C09049=1046.535,19.127,-78.806,170.149,34.517,156.500
C09050=1046.529,18.878,-78.790,170.147,34.515,156.499
C09051=1046.523,18.628,-78.775,170.146,34.514,156.499
C09052=1046.516,18.379,-78.759,170.144,34.512,156.499
C09053=1046.510,18.129,-78.743,170.142,34.511,156.499
C09054=1046.504,17.880,-78.728,170.140,34.509,156.498
C09055=1046.497,17.631,-78.712,170.139,34.508,156.498
C09056=1046.491,17.381,-78.696,170.137,34.506,156.498
C09057=1046.485,17.132,-78.681,170.135,34.505,156.498
C09058=1046.479,16.882,-78.665,170.133,34.503,156.497
C09059=1046.473,16.633,-78.650,170.132,34.502,156.497
C09060=1046.466,16.384,-78.634,170.130,34.500,156.497
C09061=1046.460,16.134,-78.618,170.128,34.499,156.497
C09062=1046.454,15.885,-78.603,170.126,34.497,156.497
C09063=1046.448,15.635,-78.587,170.124,34.495,156.496
C09064=1046.441,15.386,-78.572,170.122,34.494,156.496
C09065=1046.435,15.137,-78.556,170.120,34.493,156.496
C09066=1046.429,14.887,-78.540,170.118,34.491,156.496
C09067=1046.422,14.638,-78.525,170.117,34.489,156.495
C09068=1046.417,14.388,-78.509,170.115,34.488,156.495
C09069=1046.410,14.139,-78.493,170.113,34.486,156.495
C09070=1046.404,13.889,-78.479,170.111,34.485,156.495
C09071=1046.397,13.640,-78.463,170.110,34.484,156.494
C09072=1046.390,13.354,-78.446,170.107,34.482,156.494
C09073=1046.382,13.069,-78.428,170.105,34.480,156.494
C09074=1046.375,12.784,-78.411,170.103,34.478,156.494
C09075=1046.368,12.499,-78.393,170.101,34.477,156.493
C09076=1046.362,12.250,-78.377,170.100,34.476,156.493
C09077=1046.355,12.000,-78.362,170.098,34.474,156.493
C09078=1046.349,11.751,-78.347,170.096,34.472,156.493
C09079=1046.342,11.501,-78.331,170.094,34.471,156.492
C09080=1046.336,11.252,-78.316,170.092,34.470,156.492
C09081=1046.329,11.003,-78.301,170.091,34.468,156.492
C09082=1046.323,10.753,-78.286,170.088,34.467,156.492
C09083=1046.317,10.503,-78.270,170.086,34.466,156.492
C09084=1046.310,10.254,-78.255,170.084,34.464,156.491
C09085=1046.304,10.004,-78.240,170.082,34.462,156.491
C09086=1046.298,9.755,-78.225,170.081,34.461,156.491
C09087=1046.291,9.506,-78.209,170.079,34.460,156.491
C09088=1046.285,9.256,-78.194,170.077,34.458,156.490
C09089=1046.278,9.006,-78.179,170.075,34.457,156.490
C09090=1046.272,8.757,-78.163,170.073,34.456,156.490
C09091=1046.266,8.507,-78.148,170.072,34.454,156.490
C09092=1046.259,8.258,-78.133,170.070,34.452,156.490
C09093=1046.253,8.008,-78.118,170.068,34.451,156.489
C09094=1046.246,7.759,-78.102,170.066,34.450,156.489
C09095=1046.241,7.510,-78.088,170.064,34.448,156.489
C09096=1046.234,7.260,-78.073,170.063,34.447,156.489
C09097=1046.228,7.011,-78.058,170.061,34.446,156.488
C09098=1046.221,6.762,-78.042,170.059,34.444,156.488
C09099=1046.216,6.512,-78.027,170.057,34.442,156.488
C09100=1046.209,6.262,-78.012,170.055,34.441,156.488
C09101=1046.203,6.013,-77.997,170.054,34.440,156.488
C09102=1046.196,5.763,-77.981,170.051,34.438,156.487
C09103=1046.190,5.515,-77.967,170.049,34.437,156.487
C09104=1046.184,5.265,-77.952,170.047,34.435,156.487
C09105=1046.177,5.015,-77.937,170.045,34.433,156.487
C09106=1046.171,4.766,-77.922,170.044,34.432,156.486
C09107=1046.165,4.516,-77.907,170.042,34.431,156.486
C09108=1046.158,4.267,-77.891,170.040,34.429,156.486
C09109=1046.152,4.017,-77.876,170.038,34.428,156.486
C09110=1046.147,3.768,-77.861,170.036,34.427,156.486
C09111=1046.140,3.518,-77.846,170.035,34.425,156.485
C09112=1046.134,3.269,-77.831,170.033,34.423,156.485
C09113=1046.127,3.019,-77.816,170.031,34.422,156.485
C09114=1046.121,2.769,-77.801,170.029,34.421,156.485
C09115=1046.115,2.521,-77.786,170.027,34.419,156.484
C09116=1046.109,2.271,-77.771,170.025,34.418,156.484
C09117=1046.102,2.022,-77.756,170.024,34.417,156.484
C09118=1046.096,1.772,-77.741,170.022,34.415,156.484
C09119=1046.089,1.522,-77.726,170.020,34.413,156.484
C09120=1046.084,1.273,-77.712,170.018,34.412,156.483
C09121=1046.077,1.024,-77.697,170.016,34.410,156.483
C09122=1046.071,0.774,-77.682,170.015,34.409,156.483
C09123=1046.065,0.524,-77.666,170.012,34.408,156.483
C09124=1046.059,0.275,-77.652,170.010,34.406,156.482
C09125=1046.053,0.025,-77.637,170.008,34.404,156.482
C09126=1046.047,-0.224,-77.622,170.006,34.403,156.482
C09127=1046.040,-0.474,-77.607,170.004,34.402,156.482
C09128=1046.035,-0.723,-77.592,170.003,34.400,156.482
C09129=1046.028,-0.972,-77.577,170.001,34.399,156.481
C09130=1046.022,-1.222,-77.562,169.999,34.398,156.481
C09131=1046.015,-1.472,-77.547,169.997,34.396,156.481
C09132=1046.010,-1.721,-77.533,169.995,34.394,156.481
C09133=1046.003,-1.970,-77.518,169.993,34.393,156.480
C09134=1045.997,-2.220,-77.503,169.992,34.392,156.480
C09135=1045.991,-2.469,-77.488,169.990,34.390,156.480
C09136=1045.984,-2.752,-77.471,169.988,34.389,156.480
C09137=1045.977,-3.036,-77.454,169.986,34.387,156.479
C09138=1045.970,-3.318,-77.437,169.984,34.386,156.479
C09139=1045.963,-3.602,-77.421,169.981,34.383,156.479
C09140=1045.957,-3.852,-77.406,169.980,34.382,156.479
C09141=1045.949,-4.101,-77.392,169.978,34.381,156.479
C09142=1045.944,-4.350,-77.377,169.976,34.379,156.478
C09143=1045.938,-4.600,-77.363,169.974,34.379,156.478
C09144=1045.931,-4.850,-77.348,169.972,34.377,156.478
C09145=1045.924,-5.099,-77.333,169.969,34.376,156.478
C09146=1045.918,-5.348,-77.319,169.967,34.375,156.478
C09147=1045.912,-5.598,-77.304,169.966,34.373,156.477
C09148=1045.906,-5.848,-77.290,169.964,34.372,156.477
C09149=1045.899,-6.097,-77.276,169.962,34.371,156.477
C09150=1045.893,-6.346,-77.261,169.960,34.369,156.477
C09151=1045.886,-6.596,-77.246,169.958,34.368,156.477
C09152=1045.879,-6.845,-77.232,169.956,34.366,156.476
C09153=1045.874,-7.095,-77.218,169.954,34.365,156.476
C09154=1045.868,-7.345,-77.203,169.952,34.364,156.476
C09155=1045.861,-7.594,-77.188,169.950,34.362,156.476
C09156=1045.855,-7.843,-77.174,169.949,34.361,156.476
C09157=1045.849,-8.093,-77.160,169.947,34.360,156.475
C09158=1045.842,-8.343,-77.145,169.945,34.358,156.475
C09159=1045.836,-8.591,-77.131,169.943,34.357,156.475
C09160=1045.830,-8.842,-77.116,169.941,34.355,156.475
C09161=1045.823,-9.091,-77.101,169.939,34.354,156.475
C09162=1045.817,-9.340,-77.087,169.937,34.353,156.474
C09163=1045.810,-9.590,-77.072,169.935,34.352,156.474
C09164=1045.804,-9.840,-77.058,169.934,34.351,156.474
C09165=1045.798,-10.089,-77.044,169.932,34.349,156.474
C09166=1045.791,-10.338,-77.029,169.930,34.348,156.474
C09167=1045.786,-10.588,-77.015,169.928,34.347,156.474
C09168=1045.779,-10.838,-77.001,169.926,34.345,156.473
C09169=1045.773,-11.087,-76.987,169.924,34.344,156.473
C09170=1045.767,-11.336,-76.972,169.922,34.342,156.473
C09171=1045.760,-11.586,-76.957,169.920,34.341,156.473
C09172=1045.754,-11.835,-76.944,169.917,34.340,156.473
C09173=1045.748,-12.085,-76.929,169.916,34.338,156.472
C09174=1045.741,-12.335,-76.914,169.914,34.337,156.472
C09175=1045.736,-12.584,-76.900,169.912,34.336,156.472
C09176=1045.729,-12.834,-76.886,169.910,34.334,156.472
C09177=1045.723,-13.083,-76.872,169.908,34.333,156.471
C09178=1045.717,-13.333,-76.857,169.906,34.332,156.471
C09179=1045.711,-13.582,-76.844,169.904,34.330,156.471
C09180=1045.704,-13.832,-76.829,169.902,34.329,156.471
C09181=1045.698,-14.082,-76.815,169.900,34.328,156.471
C09182=1045.692,-14.331,-76.801,169.898,34.327,156.471
C09183=1045.685,-14.580,-76.786,169.896,34.325,156.470
C09184=1045.680,-14.830,-76.772,169.895,34.324,156.470
C09185=1045.673,-15.079,-76.758,169.893,34.323,156.470
C09186=1045.667,-15.329,-76.744,169.891,34.321,156.470
C09187=1045.661,-15.579,-76.730,169.889,34.320,156.470
C09188=1045.655,-15.828,-76.716,169.887,34.318,156.469
C09189=1045.648,-16.078,-76.702,169.885,34.318,156.469
C09190=1045.642,-16.327,-76.687,169.883,34.316,156.469
C09191=1045.635,-16.577,-76.674,169.881,34.315,156.469
C09192=1045.628,-16.826,-76.659,169.879,34.314,156.469
C09193=1045.623,-17.076,-76.645,169.877,34.312,156.468
C09194=1045.616,-17.326,-76.632,169.875,34.311,156.468
C09195=1045.610,-17.574,-76.617,169.873,34.310,156.468
C09196=1045.603,-17.824,-76.604,169.871,34.309,156.468
C09197=1045.598,-18.073,-76.589,169.869,34.307,156.468
C09198=1045.591,-18.323,-76.575,169.868,34.307,156.468
C09199=1045.585,-18.573,-76.562,169.866,34.305,156.468
C09200=1045.577,-18.854,-76.546,169.863,34.304,156.467
C09201=1045.570,-19.136,-76.530,169.861,34.302,156.467
C09202=1045.563,-19.417,-76.514,169.858,34.301,156.467
C09203=1045.556,-19.699,-76.499,169.856,34.300,156.467
C09204=1045.550,-19.949,-76.484,169.854,34.298,156.467
C09205=1045.543,-20.198,-76.471,169.852,34.297,156.466
C09206=1045.537,-20.448,-76.457,169.850,34.296,156.466
C09207=1045.531,-20.697,-76.443,169.848,34.295,156.466
C09208=1045.524,-20.947,-76.429,169.846,34.293,156.466
C09209=1045.518,-21.196,-76.415,169.844,34.292,156.466
C09210=1045.512,-21.446,-76.402,169.842,34.291,156.465
C09211=1045.506,-21.695,-76.387,169.840,34.290,156.465
C09212=1045.499,-21.945,-76.373,169.838,34.289,156.465
C09213=1045.493,-22.195,-76.360,169.836,34.287,156.465
C09214=1045.487,-22.444,-76.346,169.834,34.286,156.465
C09215=1045.480,-22.694,-76.332,169.832,34.284,156.465
C09216=1045.475,-22.943,-76.318,169.830,34.284,156.464
C09217=1045.468,-23.193,-76.304,169.828,34.282,156.464
C09218=1045.462,-23.442,-76.291,169.826,34.281,156.464
C09219=1045.455,-23.692,-76.276,169.825,34.280,156.464
C09220=1045.449,-23.941,-76.263,169.823,34.279,156.464
C09221=1045.443,-24.191,-76.250,169.821,34.277,156.464
C09222=1045.437,-24.441,-76.235,169.819,34.276,156.463
C09223=1045.431,-24.690,-76.222,169.817,34.275,156.463
C09224=1045.425,-24.940,-76.208,169.815,34.274,156.463
C09225=1045.418,-25.189,-76.194,169.813,34.273,156.463
C09226=1045.412,-25.438,-76.181,169.811,34.271,156.463
C09227=1045.406,-25.689,-76.166,169.809,34.270,156.462
C09228=1045.400,-25.938,-76.153,169.807,34.269,156.462
C09229=1045.393,-26.187,-76.140,169.805,34.268,156.462
C09230=1045.387,-26.437,-76.126,169.803,34.266,156.462
C09231=1045.381,-26.687,-76.112,169.801,34.265,156.462
C09232=1045.374,-26.935,-76.098,169.799,34.264,156.462
C09233=1045.368,-27.186,-76.084,169.797,34.263,156.462
C09234=1045.362,-27.435,-76.071,169.795,34.261,156.461
C09235=1045.355,-27.685,-76.057,169.793,34.261,156.461
C09236=1045.349,-27.934,-76.044,169.791,34.259,156.461
C09237=1045.343,-28.183,-76.031,169.789,34.259,156.461
C09238=1045.336,-28.433,-76.017,169.786,34.257,156.461
C09239=1045.330,-28.683,-76.004,169.784,34.256,156.461
C09240=1045.324,-28.932,-75.990,169.782,34.255,156.460
C09241=1045.318,-29.182,-75.976,169.780,34.254,156.460
C09242=1045.311,-29.431,-75.963,169.778,34.253,156.460
C09243=1045.305,-29.681,-75.949,169.776,34.251,156.460
C09244=1045.298,-29.931,-75.936,169.774,34.251,156.460
C09245=1045.292,-30.180,-75.923,169.772,34.249,156.460
C09246=1045.285,-30.430,-75.909,169.770,34.248,156.459
C09247=1045.279,-30.679,-75.896,169.768,34.247,156.459
C09248=1045.273,-30.929,-75.883,169.766,34.246,156.459
C09249=1045.268,-31.179,-75.870,169.764,34.245,156.459
C09250=1045.261,-31.428,-75.856,169.762,34.244,156.459
C09251=1045.255,-31.678,-75.843,169.760,34.242,156.459
C09252=1045.249,-31.927,-75.829,169.758,34.242,156.459
C09253=1045.242,-32.177,-75.816,169.756,34.240,156.458
C09254=1045.235,-32.426,-75.802,169.754,34.239,156.458
C09255=1045.229,-32.675,-75.789,169.752,34.238,156.458
C09256=1045.222,-32.925,-75.776,169.750,34.237,156.458
C09257=1045.216,-33.175,-75.762,169.748,34.236,156.458
C09258=1045.210,-33.425,-75.750,169.746,34.235,156.458
C09259=1045.204,-33.674,-75.736,169.744,34.234,156.458
C09260=1045.198,-33.924,-75.722,169.742,34.232,156.457
C09261=1045.192,-34.173,-75.709,169.740,34.232,156.457
C09262=1045.186,-34.423,-75.696,169.738,34.230,156.457
C09263=1045.179,-34.672,-75.682,169.736,34.229,156.457
C09264=1045.172,-34.953,-75.668,169.733,34.228,156.457
C09265=1045.165,-35.233,-75.653,169.731,34.227,156.457
C09266=1045.158,-35.515,-75.638,169.729,34.225,156.456
C09267=1045.151,-35.795,-75.623,169.726,34.224,156.456
C09268=1045.144,-36.045,-75.610,169.724,34.223,156.456
C09269=1045.138,-36.294,-75.596,169.722,34.222,156.456
C09270=1045.132,-36.544,-75.584,169.720,34.221,156.456
C09271=1045.126,-36.794,-75.571,169.718,34.220,156.456
C09272=1045.120,-37.043,-75.557,169.716,34.219,156.456
C09273=1045.113,-37.293,-75.544,169.714,34.217,156.455
C09274=1045.108,-37.543,-75.531,169.712,34.217,156.455
C09275=1045.102,-37.792,-75.517,169.710,34.215,156.455
C09276=1045.096,-38.042,-75.504,169.708,34.214,156.455
C09277=1045.090,-38.291,-75.492,169.706,34.213,156.455
C09278=1045.083,-38.541,-75.478,169.704,34.212,156.455
C09279=1045.077,-38.791,-75.465,169.702,34.211,156.455
C09280=1045.071,-39.041,-75.452,169.700,34.210,156.454
C09281=1045.064,-39.290,-75.439,169.698,34.209,156.454
C09282=1045.057,-39.539,-75.426,169.696,34.208,156.454
C09283=1045.051,-39.789,-75.413,169.694,34.207,156.454
C09284=1045.045,-40.039,-75.400,169.692,34.206,156.454
C09285=1045.039,-40.289,-75.387,169.689,34.205,156.454
C09286=1045.032,-40.537,-75.375,169.687,34.204,156.454
C09287=1045.026,-40.787,-75.361,169.685,34.203,156.454
C09288=1045.020,-41.037,-75.349,169.683,34.202,156.453
C09289=1045.013,-41.287,-75.335,169.681,34.201,156.453
C09290=1045.007,-41.536,-75.323,169.678,34.200,156.453
C09291=1045.001,-41.786,-75.309,169.676,34.199,156.453
C09292=1044.994,-42.035,-75.297,169.674,34.198,156.453
C09293=1044.988,-42.285,-75.284,169.672,34.197,156.453
C09294=1044.982,-42.534,-75.272,169.670,34.196,156.453
C09295=1044.976,-42.784,-75.258,169.668,34.195,156.453
C09296=1044.969,-43.034,-75.245,169.666,34.194,156.452
C09297=1044.962,-43.283,-75.233,169.663,34.193,156.452
C09298=1044.956,-43.533,-75.219,169.661,34.192,156.452
C09299=1044.950,-43.782,-75.207,169.659,34.191,156.452
C09300=1044.944,-44.032,-75.194,169.657,34.191,156.452
C09301=1044.938,-44.282,-75.181,169.655,34.189,156.452
C09302=1044.932,-44.531,-75.169,169.653,34.188,156.452
C09303=1044.925,-44.780,-75.156,169.651,34.188,156.452
C09304=1044.919,-45.030,-75.143,169.649,34.186,156.451
C09305=1044.913,-45.280,-75.130,169.647,34.185,156.451
C09306=1044.907,-45.529,-75.118,169.645,34.185,156.451
C09307=1044.900,-45.779,-75.104,169.643,34.183,156.451
C09308=1044.894,-46.029,-75.092,169.640,34.183,156.451
C09309=1044.888,-46.279,-75.079,169.638,34.182,156.451
C09310=1044.882,-46.528,-75.066,169.636,34.180,156.451
C09311=1044.875,-46.778,-75.054,169.634,34.180,156.451
C09312=1044.869,-47.027,-75.041,169.632,34.179,156.451
C09313=1044.863,-47.277,-75.028,169.630,34.177,156.450
C09314=1044.857,-47.527,-75.016,169.628,34.177,156.450
C09315=1044.850,-47.776,-75.003,169.626,34.176,156.450
C09316=1044.844,-48.026,-74.991,169.624,34.175,156.450
C09317=1044.838,-48.275,-74.978,169.622,34.174,156.450
C09318=1044.832,-48.525,-74.965,169.619,34.173,156.450
C09319=1044.825,-48.774,-74.953,169.617,34.172,156.450
C09320=1044.819,-49.024,-74.940,169.615,34.171,156.450
C09321=1044.813,-49.273,-74.927,169.613,34.170,156.450
C09322=1044.807,-49.523,-74.914,169.611,34.169,156.449
C09323=1044.801,-49.773,-74.902,169.609,34.168,156.449
C09324=1044.794,-50.022,-74.889,169.607,34.167,156.449
C09325=1044.789,-50.272,-74.877,169.605,34.166,156.449
C09326=1044.782,-50.522,-74.865,169.603,34.165,156.449
C09327=1044.776,-50.771,-74.852,169.600,34.164,156.449
C09328=1044.769,-51.053,-74.838,169.598,34.163,156.449
C09329=1044.761,-51.333,-74.824,169.596,34.163,156.449
C09330=1044.754,-51.615,-74.810,169.593,34.162,156.449
C09331=1044.747,-51.896,-74.796,169.591,34.160,156.448
C09332=1044.741,-52.146,-74.784,169.589,34.160,156.448
C09333=1044.735,-52.396,-74.772,169.586,34.159,156.448
C09334=1044.728,-52.645,-74.760,169.584,34.158,156.448
C09335=1044.722,-52.894,-74.747,169.582,34.157,156.448
C09336=1044.715,-53.144,-74.735,169.580,34.157,156.448
C09337=1044.709,-53.393,-74.723,169.578,34.156,156.448
C09338=1044.703,-53.643,-74.710,169.576,34.155,156.448
C09339=1044.696,-53.893,-74.698,169.573,34.154,156.448
C09340=1044.690,-54.143,-74.686,169.571,34.153,156.448
C09341=1044.684,-54.392,-74.674,169.569,34.153,156.448
C09342=1044.677,-54.642,-74.662,169.567,34.152,156.447
C09343=1044.671,-54.892,-74.649,169.565,34.151,156.447
C09344=1044.664,-55.141,-74.637,169.563,34.150,156.447
C09345=1044.657,-55.390,-74.625,169.560,34.150,156.447
C09346=1044.651,-55.640,-74.612,169.558,34.149,156.447
C09347=1044.645,-55.890,-74.600,169.556,34.148,156.447
C09348=1044.639,-56.140,-74.587,169.554,34.147,156.447
C09349=1044.632,-56.389,-74.576,169.552,34.147,156.447
C09350=1044.626,-56.639,-74.564,169.550,34.146,156.447
C09351=1044.620,-56.889,-74.551,169.547,34.145,156.447
C09352=1044.613,-57.138,-74.539,169.545,34.144,156.447
C09353=1044.606,-57.388,-74.527,169.543,34.143,156.447
C09354=1044.601,-57.637,-74.515,169.541,34.143,156.447
C09355=1044.594,-57.887,-74.503,169.539,34.142,156.446
C09356=1044.589,-58.137,-74.490,169.537,34.141,156.446
C09357=1044.582,-58.386,-74.478,169.534,34.140,156.446
C09358=1044.575,-58.636,-74.466,169.532,34.140,156.446
C09359=1044.570,-58.886,-74.455,169.530,34.139,156.446
C09360=1044.563,-59.136,-74.443,169.528,34.138,156.446
C09361=1044.556,-59.385,-74.431,169.526,34.137,156.446
C09362=1044.551,-59.634,-74.419,169.523,34.136,156.446
C09363=1044.544,-59.884,-74.407,169.521,34.136,156.446
C09364=1044.538,-60.134,-74.395,169.519,34.135,156.446
C09365=1044.532,-60.384,-74.382,169.517,34.134,156.446
C09366=1044.525,-60.633,-74.370,169.515,34.133,156.446
C09367=1044.519,-60.883,-74.358,169.512,34.133,156.445
C09368=1044.513,-61.132,-74.346,169.510,34.132,156.445
C09369=1044.507,-61.382,-74.335,169.508,34.131,156.445
C09370=1044.500,-61.632,-74.323,169.506,34.130,156.445
C09371=1044.494,-61.881,-74.310,169.504,34.130,156.445
C09372=1044.488,-62.131,-74.298,169.502,34.129,156.445
C09373=1044.482,-62.380,-74.287,169.499,34.128,156.445
C09374=1044.476,-62.630,-74.274,169.497,34.127,156.445
C09375=1044.469,-62.880,-74.263,169.495,34.126,156.445
C09376=1044.463,-63.130,-74.251,169.493,34.126,156.445
C09377=1044.457,-63.379,-74.238,169.491,34.125,156.445
C09378=1044.451,-63.628,-74.227,169.488,34.124,156.445
C09379=1044.444,-63.878,-74.215,169.486,34.123,156.445
C09380=1044.438,-64.128,-74.204,169.484,34.123,156.444
C09381=1044.432,-64.378,-74.191,169.482,34.122,156.444
C09382=1044.426,-64.627,-74.179,169.480,34.121,156.444
C09383=1044.419,-64.876,-74.167,169.477,34.120,156.444
C09384=1044.414,-65.127,-74.156,169.475,34.120,156.444
C09385=1044.407,-65.377,-74.144,169.473,34.119,156.444
C09386=1044.401,-65.625,-74.132,169.471,34.119,156.444
C09387=1044.395,-65.875,-74.119,169.469,34.118,156.444
C09388=1044.389,-66.125,-74.108,169.466,34.117,156.444
C09389=1044.383,-66.374,-74.097,169.464,34.116,156.444
C09390=1044.376,-66.624,-74.085,169.462,34.115,156.444
C09391=1044.370,-66.874,-74.073,169.460,34.115,156.444
C09392=1044.364,-67.122,-74.062,169.457,34.114,156.444
C09393=1044.358,-67.370,-74.049,169.455,34.113,156.444
C09394=1044.352,-67.618,-74.038,169.453,34.112,156.443
C09395=1044.346,-67.865,-74.026,169.451,34.112,156.443
C09396=1044.339,-68.113,-74.014,169.449,34.111,156.443
C09397=1044.334,-68.362,-74.003,169.447,34.111,156.443
C09398=1044.327,-68.610,-73.991,169.444,34.110,156.443
C09399=1044.321,-68.857,-73.979,169.442,34.109,156.443
C09400=1044.315,-69.108,-73.968,169.440,34.108,156.443
C09401=1044.309,-69.356,-73.956,169.438,34.108,156.443
C09402=1044.303,-69.607,-73.945,169.435,34.107,156.443
C09403=1044.297,-69.855,-73.933,169.433,34.107,156.443
C09404=1044.291,-70.105,-73.921,169.431,34.106,156.443
C09405=1044.285,-70.356,-73.909,169.429,34.105,156.443
C09406=1044.279,-70.604,-73.898,169.427,34.104,156.443
C09407=1044.272,-70.855,-73.887,169.424,34.103,156.443
C09408=1044.267,-71.104,-73.874,169.422,34.103,156.443
C09409=1044.261,-71.354,-73.863,169.420,34.102,156.442
C09410=1044.254,-71.604,-73.851,169.418,34.102,156.442
C09411=1044.248,-71.853,-73.840,169.415,34.101,156.442
C09412=1044.242,-72.103,-73.828,169.413,34.100,156.442
C09413=1044.237,-72.352,-73.817,169.411,34.099,156.442
C09414=1044.230,-72.602,-73.805,169.409,34.099,156.442
C09415=1044.224,-72.852,-73.794,169.407,34.098,156.442
C09416=1044.218,-73.101,-73.782,169.404,34.098,156.442
C09417=1044.212,-73.352,-73.770,169.402,34.097,156.442
C09418=1044.206,-73.600,-73.759,169.400,34.096,156.442
C09419=1044.200,-73.851,-73.747,169.398,34.095,156.442
C09420=1044.194,-74.099,-73.736,169.395,34.095,156.442
C09421=1044.187,-74.350,-73.725,169.393,34.094,156.442
C09422=1044.181,-74.599,-73.714,169.391,34.094,156.442
C09423=1044.175,-74.849,-73.702,169.389,34.093,156.442
C09424=1044.168,-75.135,-73.688,169.386,34.093,156.442
C09425=1044.161,-75.421,-73.676,169.383,34.092,156.442
C09426=1044.153,-75.707,-73.663,169.381,34.091,156.442
C09427=1044.146,-75.993,-73.650,169.378,34.090,156.442
C09428=1044.140,-76.243,-73.639,169.376,34.090,156.442
C09429=1044.134,-76.493,-73.627,169.374,34.089,156.441
C09430=1044.128,-76.742,-73.616,169.371,34.089,156.442
C09431=1044.121,-76.992,-73.605,169.369,34.088,156.441
C09432=1044.116,-77.241,-73.594,169.367,34.088,156.441
C09433=1044.109,-77.491,-73.582,169.365,34.088,156.441
C09434=1044.103,-77.740,-73.571,169.362,34.087,156.441
C09435=1044.097,-77.991,-73.560,169.360,34.086,156.441
C09436=1044.091,-78.240,-73.549,169.358,34.086,156.441
C09437=1044.085,-78.490,-73.537,169.355,34.085,156.441
C09438=1044.079,-78.739,-73.526,169.353,34.085,156.441
C09439=1044.073,-78.989,-73.515,169.351,34.084,156.441
C09440=1044.067,-79.239,-73.504,169.349,34.084,156.441
C09441=1044.060,-79.488,-73.492,169.346,34.083,156.441
C09442=1044.054,-79.738,-73.481,169.344,34.082,156.441
C09443=1044.047,-79.988,-73.470,169.342,34.082,156.441
C09444=1044.042,-80.237,-73.460,169.339,34.081,156.441
C09445=1044.035,-80.488,-73.448,169.337,34.081,156.441
C09446=1044.030,-80.737,-73.437,169.335,34.081,156.441
C09447=1044.022,-80.986,-73.426,169.333,34.080,156.441
C09448=1044.016,-81.236,-73.415,169.330,34.080,156.441
C09449=1044.010,-81.486,-73.404,169.328,34.079,156.441
C09450=1044.004,-81.735,-73.394,169.326,34.079,156.441
C09451=1043.997,-81.985,-73.382,169.324,34.079,156.441
C09452=1043.991,-82.235,-73.371,169.322,34.078,156.441
C09453=1043.984,-82.485,-73.361,169.320,34.078,156.441
C09454=1043.979,-82.734,-73.350,169.317,34.077,156.441
C09455=1043.972,-82.984,-73.339,169.315,34.077,156.441
C09456=1043.965,-83.268,-73.326,169.312,34.076,156.441
C09457=1043.958,-83.554,-73.314,169.310,34.076,156.441
C09458=1043.951,-83.838,-73.301,169.307,34.076,156.441
C09459=1043.944,-84.123,-73.289,169.304,34.075,156.441
C09460=1043.938,-84.373,-73.278,169.302,34.075,156.441
C09461=1043.931,-84.623,-73.267,169.300,34.074,156.441
C09462=1043.925,-84.872,-73.256,169.298,34.074,156.441
C09463=1043.919,-85.122,-73.245,169.295,34.074,156.441
C09464=1043.912,-85.371,-73.235,169.293,34.073,156.441
C09465=1043.907,-85.621,-73.224,169.291,34.073,156.441
C09466=1043.900,-85.871,-73.213,169.288,34.073,156.441
C09467=1043.894,-86.120,-73.202,169.286,34.072,156.441
C09468=1043.887,-86.370,-73.191,169.284,34.072,156.441
C09469=1043.882,-86.620,-73.180,169.281,34.072,156.441
C09470=1043.875,-86.869,-73.170,169.279,34.071,156.441
C09471=1043.869,-87.119,-73.159,169.277,34.071,156.441
C09472=1043.863,-87.369,-73.148,169.274,34.071,156.441
C09473=1043.857,-87.618,-73.138,169.272,34.070,156.441
C09474=1043.850,-87.868,-73.126,169.270,34.070,156.441
C09475=1043.845,-88.118,-73.116,169.267,34.070,156.441
C09476=1043.838,-88.368,-73.106,169.265,34.069,156.441
C09477=1043.832,-88.618,-73.095,169.263,34.069,156.441
C09478=1043.826,-88.867,-73.084,169.260,34.068,156.441
C09479=1043.819,-89.117,-73.073,169.258,34.068,156.441
C09480=1043.813,-89.366,-73.062,169.256,34.068,156.441
C09481=1043.808,-89.616,-73.051,169.253,34.067,156.441
C09482=1043.801,-89.865,-73.041,169.251,34.067,156.441
C09483=1043.795,-90.116,-73.031,169.249,34.066,156.441
C09484=1043.789,-90.365,-73.020,169.246,34.066,156.441
C09485=1043.783,-90.615,-73.010,169.244,34.066,156.441
C09486=1043.777,-90.865,-72.998,169.242,34.065,156.441
C09487=1043.770,-91.114,-72.988,169.239,34.065,156.441
C09488=1043.765,-91.364,-72.978,169.237,34.065,156.441
C09489=1043.758,-91.614,-72.967,169.235,34.065,156.441
C09490=1043.752,-91.863,-72.956,169.232,34.064,156.441
C09491=1043.746,-92.113,-72.945,169.230,34.064,156.441
C09492=1043.740,-92.362,-72.935,169.228,34.064,156.441
C09493=1043.734,-92.613,-72.925,169.225,34.064,156.441
C09494=1043.728,-92.862,-72.914,169.223,34.063,156.441
C09495=1043.721,-93.112,-72.903,169.221,34.063,156.441
C09496=1043.716,-93.361,-72.893,169.218,34.063,156.441
C09497=1043.709,-93.612,-72.883,169.216,34.062,156.441
C09498=1043.703,-93.861,-72.872,169.214,34.062,156.441
C09499=1043.697,-94.111,-72.861,169.211,34.061,156.441
C09500=1043.691,-94.360,-72.851,169.209,34.061,156.441
C09501=1043.686,-94.610,-72.840,169.206,34.061,156.441
C09502=1043.678,-94.860,-72.830,169.204,34.061,156.441
C09503=1043.673,-95.110,-72.820,169.202,34.060,156.441
C09504=1043.667,-95.359,-72.809,169.199,34.060,156.441
C09505=1043.661,-95.609,-72.798,169.197,34.060,156.441
C09506=1043.655,-95.859,-72.788,169.196,34.060,156.441
C09507=1043.648,-96.109,-72.778,169.193,34.060,156.441
C09508=1043.643,-96.358,-72.767,169.191,34.059,156.441
C09509=1043.636,-96.608,-72.757,169.189,34.059,156.441
C09510=1043.631,-96.857,-72.746,169.186,34.058,156.441
C09511=1043.625,-97.107,-72.735,169.184,34.058,156.441
C09512=1043.619,-97.357,-72.726,169.182,34.058,156.441
C09513=1043.612,-97.607,-72.715,169.179,34.058,156.441
C09514=1043.606,-97.857,-72.705,169.177,34.058,156.441
C09515=1043.600,-98.106,-72.695,169.175,34.058,156.441
C09516=1043.594,-98.356,-72.685,169.172,34.058,156.441
C09517=1043.588,-98.605,-72.674,169.170,34.057,156.441
C09518=1043.582,-98.855,-72.665,169.167,34.057,156.441
C09519=1043.575,-99.105,-72.654,169.165,34.057,156.441
C09520=1043.569,-99.392,-72.643,169.162,34.057,156.441
C09521=1043.561,-99.678,-72.631,169.159,34.057,156.441
C09522=1043.554,-99.966,-72.619,169.157,34.057,156.442
C09523=1043.547,-100.253,-72.607,169.154,34.056,156.442
C09524=1043.541,-100.502,-72.597,169.152,34.056,156.442
C09525=1043.535,-100.753,-72.587,169.149,34.056,156.442
C09526=1043.529,-101.002,-72.577,169.147,34.056,156.442
C09527=1043.523,-101.252,-72.567,169.144,34.056,156.442
C09528=1043.516,-101.502,-72.556,169.142,34.056,156.442
C09529=1043.510,-101.752,-72.547,169.140,34.055,156.442
C09530=1043.504,-102.001,-72.536,169.137,34.055,156.442
C09531=1043.498,-102.251,-72.526,169.135,34.055,156.442
C09532=1043.492,-102.501,-72.517,169.133,34.055,156.442
C09533=1043.485,-102.750,-72.506,169.130,34.055,156.442
C09534=1043.479,-103.000,-72.497,169.128,34.055,156.442
C09535=1043.474,-103.249,-72.486,169.125,34.054,156.442
C09536=1043.467,-103.499,-72.476,169.123,34.054,156.442
C09537=1043.461,-103.749,-72.467,169.121,34.054,156.442
C09538=1043.455,-103.998,-72.456,169.118,34.055,156.442
C09539=1043.449,-104.248,-72.446,169.116,34.055,156.442
C09540=1043.443,-104.498,-72.436,169.113,34.054,156.442
C09541=1043.436,-104.748,-72.426,169.111,34.054,156.442
C09542=1043.431,-104.998,-72.416,169.109,34.054,156.442
C09543=1043.424,-105.248,-72.406,169.106,34.054,156.442
C09544=1043.418,-105.497,-72.397,169.104,34.054,156.442
C09545=1043.412,-105.747,-72.386,169.102,34.054,156.442
C09546=1043.406,-105.997,-72.376,169.100,34.054,156.443
C09547=1043.400,-106.246,-72.367,169.098,34.054,156.443
C09548=1043.394,-106.496,-72.356,169.095,34.054,156.443
C09549=1043.388,-106.745,-72.347,169.093,34.054,156.443
C09550=1043.382,-106.996,-72.337,169.090,34.053,156.443
C09551=1043.376,-107.245,-72.327,169.088,34.053,156.443
C09552=1043.370,-107.495,-72.318,169.086,34.054,156.443
C09553=1043.363,-107.744,-72.307,169.083,34.054,156.443
C09554=1043.357,-107.994,-72.298,169.081,34.053,156.443
C09555=1043.351,-108.244,-72.288,169.078,34.053,156.443
C09556=1043.345,-108.494,-72.279,169.076,34.054,156.443
C09557=1043.339,-108.743,-72.269,169.073,34.054,156.443
C09558=1043.333,-108.994,-72.259,169.071,34.053,156.443
C09559=1043.327,-109.243,-72.249,169.069,34.053,156.443
C09560=1043.321,-109.493,-72.239,169.066,34.054,156.443
C09561=1043.314,-109.742,-72.229,169.064,34.054,156.444
C09562=1043.308,-109.992,-72.220,169.061,34.053,156.444
C09563=1043.302,-110.242,-72.210,169.059,34.054,156.444
C09564=1043.296,-110.492,-72.201,169.056,34.054,156.444
C09565=1043.290,-110.742,-72.191,169.054,34.054,156.444
C09566=1043.283,-110.991,-72.182,169.052,34.054,156.444
C09567=1043.277,-111.241,-72.172,169.049,34.054,156.444
C09568=1043.271,-111.490,-72.162,169.047,34.054,156.444
C09569=1043.265,-111.739,-72.153,169.044,34.054,156.444
C09570=1043.260,-111.990,-72.142,169.042,34.054,156.444
C09571=1043.254,-112.239,-72.133,169.039,34.054,156.444
C09572=1043.247,-112.489,-72.123,169.037,34.054,156.444
C09573=1043.241,-112.739,-72.114,169.035,34.054,156.444
C09574=1043.235,-112.989,-72.104,169.032,34.054,156.444
C09575=1043.229,-113.239,-72.095,169.030,34.055,156.445
C09576=1043.223,-113.488,-72.085,169.028,34.054,156.445
C09577=1043.217,-113.738,-72.075,169.026,34.054,156.445
C09578=1043.210,-113.988,-72.066,169.023,34.055,156.445
C09579=1043.204,-114.238,-72.056,169.021,34.055,156.445
C09580=1043.199,-114.487,-72.047,169.019,34.054,156.445
C09581=1043.193,-114.737,-72.038,169.016,34.055,156.445
C09582=1043.186,-114.986,-72.028,169.014,34.055,156.445
C09583=1043.180,-115.236,-72.018,169.011,34.055,156.445
C09584=1043.173,-115.523,-72.008,169.008,34.055,156.445
C09585=1043.166,-115.809,-71.997,169.006,34.056,156.445
C09586=1043.160,-116.094,-71.986,169.003,34.055,156.445
C09587=1043.152,-116.381,-71.976,169.000,34.056,156.446
C09588=1043.146,-116.630,-71.966,168.998,34.056,156.446
C09589=1043.140,-116.880,-71.957,168.995,34.056,156.446
C09590=1043.134,-117.130,-71.947,168.993,34.056,156.446
C09591=1043.128,-117.379,-71.938,168.990,34.056,156.446
C09592=1043.122,-117.630,-71.929,168.988,34.056,156.446
C09593=1043.116,-117.879,-71.919,168.985,34.057,156.446
C09594=1043.110,-118.129,-71.910,168.983,34.057,156.446
C09595=1043.103,-118.379,-71.901,168.980,34.057,156.446
C09596=1043.097,-118.628,-71.891,168.978,34.057,156.446
C09597=1043.091,-118.878,-71.882,168.976,34.057,156.447
C09598=1043.085,-119.128,-71.873,168.973,34.057,156.447
C09599=1043.079,-119.378,-71.864,168.971,34.058,156.447
C09600=1043.073,-119.628,-71.854,168.968,34.058,156.447
C09601=1043.067,-119.877,-71.845,168.966,34.058,156.447
C09602=1043.062,-120.127,-71.836,168.963,34.059,156.447
C09603=1043.055,-120.377,-71.827,168.962,34.058,156.447
C09604=1043.048,-120.626,-71.818,168.959,34.059,156.447
C09605=1043.042,-120.876,-71.808,168.957,34.059,156.447
C09606=1043.037,-121.126,-71.799,168.954,34.059,156.447
C09607=1043.031,-121.376,-71.790,168.952,34.060,156.448
C09608=1043.025,-121.625,-71.780,168.949,34.060,156.448
C09609=1043.018,-121.876,-71.772,168.947,34.060,156.448
C09610=1043.013,-122.125,-71.763,168.945,34.061,156.448
C09611=1043.006,-122.374,-71.753,168.942,34.060,156.448
C09612=1043.000,-122.624,-71.744,168.940,34.061,156.448
C09613=1042.994,-122.875,-71.735,168.937,34.061,156.448
C09614=1042.989,-123.124,-71.726,168.935,34.061,156.448
C09615=1042.982,-123.373,-71.717,168.932,34.062,156.448
C09616=1042.976,-123.624,-71.708,168.930,34.062,156.448
C09617=1042.970,-123.874,-71.698,168.927,34.062,156.449
C09618=1042.965,-124.123,-71.690,168.925,34.062,156.449
C09619=1042.958,-124.373,-71.680,168.922,34.062,156.449
C09620=1042.951,-124.622,-71.671,168.920,34.063,156.449
C09621=1042.946,-124.872,-71.663,168.917,34.063,156.449
C09622=1042.940,-125.122,-71.653,168.915,34.064,156.449
C09623=1042.933,-125.372,-71.645,168.912,34.064,156.449
C09624=1042.927,-125.622,-71.635,168.910,34.064,156.449
C09625=1042.922,-125.872,-71.627,168.907,34.065,156.450
C09626=1042.915,-126.121,-71.618,168.905,34.065,156.450
C09627=1042.909,-126.371,-71.608,168.903,34.065,156.450
C09628=1042.904,-126.621,-71.600,168.901,34.065,156.450
C09629=1042.897,-126.870,-71.591,168.899,34.066,156.450
C09630=1042.891,-127.121,-71.582,168.896,34.066,156.450
C09631=1042.885,-127.370,-71.573,168.894,34.066,156.450
C09632=1042.879,-127.620,-71.565,168.891,34.067,156.450
C09633=1042.873,-127.869,-71.555,168.889,34.067,156.450
C09634=1042.868,-128.119,-71.545,168.886,34.067,156.451
C09635=1042.864,-128.369,-71.536,168.884,34.066,156.450
C09636=1042.860,-128.619,-71.525,168.882,34.065,156.450
C09637=1042.858,-128.869,-71.514,168.880,34.064,156.450
C09638=1042.856,-129.118,-71.501,168.878,34.062,156.450
C09639=1042.856,-129.368,-71.489,168.877,34.059,156.449
C09640=1042.856,-129.619,-71.476,168.875,34.057,156.449
C09641=1042.857,-129.869,-71.462,168.873,34.053,156.449
C09642=1042.858,-130.119,-71.447,168.871,34.049,156.448
C09643=1042.860,-130.369,-71.433,168.870,34.045,156.447
C09644=1042.864,-130.619,-71.417,168.869,34.040,156.446
C09645=1042.869,-130.869,-71.401,168.868,34.036,156.446
C09646=1042.874,-131.120,-71.384,168.867,34.030,156.445
C09647=1042.880,-131.370,-71.367,168.867,34.023,156.444
C09648=1042.529,-131.394,-71.617,168.820,34.211,156.477
C09649=1042.523,-131.144,-71.635,168.821,34.218,156.478
C09650=1042.518,-130.894,-71.651,168.821,34.223,156.479
C09651=1042.512,-130.644,-71.667,168.822,34.228,156.479
C09652=1042.510,-130.392,-71.683,168.823,34.233,156.480
C09653=1042.507,-130.143,-71.697,168.824,34.237,156.481
C09654=1042.505,-129.893,-71.712,168.827,34.241,156.482
C09655=1042.504,-129.643,-71.726,168.828,34.244,156.482
C09656=1042.504,-129.392,-71.739,168.830,34.247,156.483
C09657=1042.505,-129.143,-71.752,168.831,34.250,156.483
C09658=1042.506,-128.893,-71.764,168.833,34.251,156.483
C09659=1042.509,-128.642,-71.776,168.835,34.253,156.483
C09660=1042.512,-128.392,-71.787,168.837,34.254,156.484
C09661=1042.516,-128.143,-71.797,168.840,34.255,156.484
C09662=1042.522,-127.893,-71.806,168.842,34.255,156.484
C09663=1042.527,-127.644,-71.815,168.844,34.254,156.483
C09664=1042.533,-127.394,-71.824,168.847,34.254,156.483
C09665=1042.539,-127.144,-71.833,168.849,34.254,156.483
C09666=1042.546,-126.895,-71.842,168.852,34.254,156.483
C09667=1042.551,-126.644,-71.851,168.854,34.253,156.483
C09668=1042.558,-126.395,-71.860,168.857,34.253,156.483
C09669=1042.564,-126.145,-71.868,168.859,34.252,156.483
C09670=1042.570,-125.895,-71.878,168.861,34.252,156.483
C09671=1042.576,-125.645,-71.887,168.863,34.252,156.482
C09672=1042.582,-125.396,-71.895,168.866,34.251,156.482
C09673=1042.588,-125.146,-71.905,168.868,34.251,156.482
C09674=1042.594,-124.896,-71.914,168.871,34.250,156.482
C09675=1042.600,-124.647,-71.922,168.873,34.250,156.482
C09676=1042.606,-124.397,-71.931,168.876,34.250,156.482
C09677=1042.612,-124.147,-71.941,168.878,34.249,156.482
C09678=1042.618,-123.897,-71.949,168.881,34.249,156.482
C09679=1042.625,-123.648,-71.958,168.883,34.249,156.482
C09680=1042.631,-123.398,-71.968,168.886,34.249,156.481
C09681=1042.637,-123.148,-71.976,168.888,34.248,156.481
C09682=1042.642,-122.899,-71.986,168.891,34.248,156.481
C09683=1042.648,-122.649,-71.995,168.893,34.248,156.481
C09684=1042.655,-122.399,-72.004,168.896,34.247,156.481
C09685=1042.661,-122.149,-72.013,168.898,34.247,156.481
C09686=1042.667,-121.900,-72.022,168.901,34.247,156.481
C09687=1042.673,-121.649,-72.031,168.903,34.246,156.481
C09688=1042.679,-121.400,-72.041,168.906,34.247,156.481
C09689=1042.685,-121.150,-72.050,168.908,34.246,156.480
C09690=1042.691,-120.901,-72.059,168.910,34.245,156.480
C09691=1042.697,-120.651,-72.068,168.913,34.246,156.480
C09692=1042.703,-120.401,-72.077,168.915,34.245,156.480
C09693=1042.709,-120.151,-72.087,168.918,34.245,156.480
C09694=1042.715,-119.901,-72.096,168.920,34.245,156.480
C09695=1042.721,-119.651,-72.105,168.922,34.244,156.480
C09696=1042.727,-119.402,-72.114,168.924,34.244,156.480
C09697=1042.734,-119.152,-72.123,168.927,34.244,156.480
C09698=1042.740,-118.902,-72.133,168.929,34.244,156.480
C09699=1042.746,-118.652,-72.142,168.932,34.244,156.479
C09700=1042.752,-118.403,-72.151,168.934,34.243,156.479
C09701=1042.758,-118.153,-72.161,168.937,34.243,156.479
C09702=1042.764,-117.903,-72.170,168.939,34.243,156.479
C09703=1042.770,-117.653,-72.180,168.942,34.243,156.479
C09704=1042.776,-117.404,-72.189,168.944,34.242,156.479
C09705=1042.781,-117.154,-72.198,168.946,34.243,156.479
C09706=1042.788,-116.904,-72.207,168.949,34.242,156.479
C09707=1042.795,-116.655,-72.216,168.951,34.242,156.479
C09708=1042.801,-116.405,-72.226,168.954,34.242,156.479
C09709=1042.807,-116.118,-72.237,168.957,34.242,156.479
C09710=1042.815,-115.833,-72.247,168.960,34.241,156.478
C09711=1042.821,-115.547,-72.258,168.962,34.241,156.478
C09712=1042.828,-115.260,-72.269,168.965,34.241,156.478
C09713=1042.834,-115.010,-72.279,168.968,34.241,156.478
C09714=1042.840,-114.760,-72.288,168.970,34.241,156.478
C09715=1042.847,-114.511,-72.297,168.973,34.240,156.478
C09716=1042.853,-114.261,-72.307,168.975,34.240,156.478
C09717=1042.859,-114.012,-72.316,168.977,34.241,156.478
C09718=1042.864,-113.762,-72.326,168.980,34.240,156.478
C09719=1042.871,-113.512,-72.336,168.982,34.240,156.478
C09720=1042.877,-113.262,-72.345,168.985,34.240,156.477
C09721=1042.883,-113.013,-72.355,168.987,34.240,156.477
C09722=1042.889,-112.763,-72.364,168.989,34.240,156.477
C09723=1042.895,-112.513,-72.374,168.991,34.240,156.477
C09724=1042.901,-112.263,-72.384,168.994,34.240,156.477
C09725=1042.908,-112.013,-72.393,168.996,34.240,156.477
C09726=1042.914,-111.764,-72.403,168.998,34.239,156.477
C09727=1042.920,-111.514,-72.412,169.001,34.239,156.477
C09728=1042.926,-111.265,-72.422,169.003,34.239,156.477
C09729=1042.932,-111.015,-72.431,169.006,34.239,156.477
C09730=1042.938,-110.765,-72.441,169.008,34.239,156.477
C09731=1042.944,-110.516,-72.451,169.011,34.239,156.477
C09732=1042.951,-110.266,-72.460,169.013,34.239,156.477
C09733=1042.956,-110.016,-72.471,169.015,34.239,156.477
C09734=1042.962,-109.766,-72.480,169.018,34.239,156.476
C09735=1042.968,-109.516,-72.490,169.020,34.239,156.476
C09736=1042.975,-109.267,-72.499,169.023,34.239,156.476
C09737=1042.981,-109.017,-72.509,169.025,34.238,156.476
C09738=1042.987,-108.767,-72.518,169.028,34.239,156.476
C09739=1042.993,-108.518,-72.529,169.030,34.239,156.476
C09740=1042.999,-108.268,-72.538,169.033,34.238,156.476
C09741=1043.006,-108.018,-72.548,169.035,34.238,156.476
C09742=1043.012,-107.768,-72.557,169.037,34.238,156.476
C09743=1043.017,-107.518,-72.568,169.040,34.239,156.476
C09744=1043.023,-107.269,-72.577,169.042,34.238,156.476
C09745=1043.030,-107.019,-72.587,169.045,34.238,156.476
C09746=1043.036,-106.770,-72.597,169.047,34.238,156.476
C09747=1043.042,-106.520,-72.607,169.050,34.239,156.476
C09748=1043.048,-106.270,-72.617,169.052,34.239,156.476
C09749=1043.054,-106.020,-72.627,169.054,34.238,156.475
C09750=1043.060,-105.771,-72.637,169.057,34.238,156.475
C09751=1043.067,-105.521,-72.646,169.059,34.238,156.475
C09752=1043.072,-105.271,-72.656,169.062,34.239,156.475
C09753=1043.078,-105.022,-72.667,169.064,34.239,156.475
C09754=1043.085,-104.772,-72.676,169.066,34.239,156.475
C09755=1043.091,-104.522,-72.686,169.068,34.238,156.475
C09756=1043.097,-104.273,-72.697,169.070,34.239,156.475
C09757=1043.103,-104.022,-72.707,169.073,34.239,156.475
C09758=1043.109,-103.772,-72.716,169.075,34.239,156.475
C09759=1043.116,-103.523,-72.726,169.077,34.239,156.475
C09760=1043.121,-103.273,-72.737,169.080,34.239,156.475
C09761=1043.128,-103.023,-72.746,169.082,34.239,156.475
C09762=1043.134,-102.774,-72.756,169.085,34.239,156.475
C09763=1043.139,-102.524,-72.767,169.087,34.239,156.475
C09764=1043.146,-102.275,-72.777,169.090,34.239,156.475
C09765=1043.152,-102.025,-72.786,169.092,34.239,156.475
C09766=1043.158,-101.775,-72.796,169.094,34.239,156.475
C09767=1043.164,-101.526,-72.807,169.097,34.240,156.475
C09768=1043.170,-101.276,-72.816,169.099,34.240,156.475
C09769=1043.177,-101.026,-72.827,169.102,34.240,156.475
C09770=1043.183,-100.776,-72.837,169.104,34.240,156.475
C09771=1043.189,-100.527,-72.848,169.106,34.240,156.475
C09772=1043.195,-100.277,-72.857,169.109,34.240,156.474
C09773=1043.202,-99.989,-72.869,169.111,34.240,156.474
C09774=1043.210,-99.702,-72.881,169.114,34.240,156.474
C09775=1043.216,-99.416,-72.892,169.117,34.240,156.474
C09776=1043.223,-99.129,-72.904,169.120,34.240,156.474
C09777=1043.229,-98.879,-72.914,169.122,34.240,156.474
C09778=1043.236,-98.629,-72.925,169.125,34.241,156.474
C09779=1043.242,-98.379,-72.935,169.127,34.241,156.474
C09780=1043.248,-98.130,-72.945,169.129,34.241,156.474
C09781=1043.254,-97.880,-72.955,169.132,34.241,156.474
C09782=1043.260,-97.631,-72.965,169.134,34.241,156.474
C09783=1043.267,-97.380,-72.975,169.136,34.241,156.474
C09784=1043.273,-97.131,-72.986,169.139,34.241,156.474
C09785=1043.279,-96.881,-72.997,169.141,34.242,156.474
C09786=1043.285,-96.631,-73.007,169.144,34.242,156.474
C09787=1043.290,-96.382,-73.018,169.146,34.242,156.474
C09788=1043.297,-96.132,-73.027,169.148,34.243,156.474
C09789=1043.303,-95.882,-73.038,169.151,34.243,156.474
C09790=1043.309,-95.633,-73.049,169.153,34.243,156.474
C09791=1043.315,-95.383,-73.059,169.155,34.243,156.474
C09792=1043.321,-95.133,-73.069,169.158,34.244,156.474
C09793=1043.327,-94.884,-73.080,169.160,34.244,156.474
C09794=1043.332,-94.634,-73.090,169.162,34.244,156.474
C09795=1043.340,-94.384,-73.101,169.165,34.244,156.474
C09796=1043.345,-94.134,-73.112,169.166,34.244,156.474
C09797=1043.351,-93.885,-73.121,169.169,34.245,156.474
C09798=1043.357,-93.635,-73.132,169.171,34.245,156.474
C09799=1043.363,-93.385,-73.143,169.173,34.245,156.474
C09800=1043.370,-93.136,-73.154,169.176,34.246,156.474
C09801=1043.375,-92.886,-73.164,169.178,34.246,156.474
C09802=1043.382,-92.636,-73.174,169.180,34.246,156.474
C09803=1043.388,-92.386,-73.185,169.183,34.247,156.474
C09804=1043.394,-92.137,-73.196,169.185,34.247,156.474
C09805=1043.400,-91.887,-73.206,169.187,34.247,156.474
C09806=1043.406,-91.638,-73.217,169.190,34.247,156.474
C09807=1043.413,-91.388,-73.227,169.192,34.248,156.474
C09808=1043.419,-91.138,-73.238,169.194,34.248,156.474
C09809=1043.424,-90.888,-73.248,169.197,34.248,156.474
C09810=1043.431,-90.639,-73.259,169.199,34.248,156.474
C09811=1043.437,-90.389,-73.270,169.201,34.248,156.474
C09812=1043.443,-90.139,-73.281,169.204,34.249,156.474
C09813=1043.449,-89.890,-73.291,169.206,34.249,156.474
C09814=1043.456,-89.640,-73.302,169.209,34.250,156.474
C09815=1043.462,-89.390,-73.312,169.211,34.250,156.474
C09816=1043.467,-89.141,-73.323,169.213,34.250,156.474
C09817=1043.474,-88.890,-73.334,169.216,34.251,156.474
C09818=1043.480,-88.641,-73.344,169.218,34.251,156.474
C09819=1043.486,-88.392,-73.355,169.220,34.251,156.474
C09820=1043.492,-88.141,-73.366,169.223,34.252,156.474
C09821=1043.499,-87.892,-73.377,169.225,34.252,156.474
C09822=1043.505,-87.643,-73.388,169.227,34.252,156.474
C09823=1043.511,-87.393,-73.399,169.230,34.253,156.474
C09824=1043.517,-87.143,-73.409,169.232,34.253,156.474
C09825=1043.523,-86.893,-73.419,169.234,34.253,156.474
C09826=1043.529,-86.643,-73.430,169.237,34.253,156.474
C09827=1043.536,-86.394,-73.441,169.239,34.254,156.474
C09828=1043.542,-86.144,-73.452,169.241,34.254,156.474
C09829=1043.548,-85.894,-73.463,169.244,34.254,156.474
C09830=1043.554,-85.645,-73.473,169.246,34.255,156.474
C09831=1043.560,-85.395,-73.484,169.248,34.255,156.474
C09832=1043.566,-85.145,-73.495,169.251,34.255,156.474
C09833=1043.573,-84.896,-73.506,169.253,34.256,156.474
C09834=1043.579,-84.646,-73.517,169.255,34.256,156.474
C09835=1043.585,-84.397,-73.528,169.258,34.256,156.474
C09836=1043.592,-84.147,-73.538,169.260,34.257,156.474
C09837=1043.599,-83.863,-73.551,169.263,34.257,156.474
C09838=1043.606,-83.577,-73.563,169.265,34.257,156.474
C09839=1043.613,-83.293,-73.575,169.268,34.258,156.474
C09840=1043.621,-83.008,-73.588,169.271,34.258,156.474
C09841=1043.626,-82.758,-73.599,169.273,34.259,156.474
C09842=1043.633,-82.508,-73.610,169.275,34.259,156.474
C09843=1043.638,-82.259,-73.621,169.278,34.259,156.474
C09844=1043.645,-82.009,-73.632,169.280,34.260,156.474
C09845=1043.651,-81.759,-73.643,169.282,34.260,156.474
C09846=1043.658,-81.509,-73.654,169.285,34.261,156.474
C09847=1043.664,-81.260,-73.664,169.287,34.261,156.474
C09848=1043.671,-81.010,-73.676,169.289,34.261,156.474
C09849=1043.676,-80.761,-73.687,169.291,34.262,156.474
C09850=1043.683,-80.511,-73.698,169.294,34.262,156.474
C09851=1043.689,-80.262,-73.709,169.296,34.262,156.474
C09852=1043.696,-80.011,-73.720,169.298,34.263,156.474
C09853=1043.701,-79.762,-73.731,169.301,34.263,156.474
C09854=1043.708,-79.512,-73.743,169.303,34.264,156.474
C09855=1043.714,-79.263,-73.754,169.305,34.264,156.474
C09856=1043.720,-79.013,-73.765,169.308,34.265,156.474
C09857=1043.726,-78.763,-73.776,169.310,34.265,156.474
C09858=1043.733,-78.513,-73.786,169.312,34.266,156.474
C09859=1043.739,-78.264,-73.798,169.314,34.266,156.474
C09860=1043.745,-78.014,-73.809,169.317,34.267,156.474
C09861=1043.751,-77.765,-73.820,169.319,34.267,156.474
C09862=1043.758,-77.515,-73.832,169.321,34.268,156.474
C09863=1043.764,-77.265,-73.843,169.324,34.269,156.474
C09864=1043.770,-77.015,-73.854,169.326,34.269,156.474
C09865=1043.776,-76.765,-73.865,169.328,34.269,156.474
C09866=1043.782,-76.516,-73.877,169.330,34.270,156.474
C09867=1043.788,-76.266,-73.888,169.333,34.270,156.474
C09868=1043.794,-76.017,-73.899,169.334,34.271,156.474
C09869=1043.801,-75.767,-73.911,169.336,34.271,156.474
C09870=1043.807,-75.518,-73.922,169.339,34.272,156.474
C09871=1043.813,-75.267,-73.933,169.341,34.272,156.474
C09872=1043.820,-75.018,-73.945,169.343,34.273,156.474
C09873=1043.825,-74.768,-73.956,169.345,34.273,156.474
C09874=1043.832,-74.519,-73.968,169.348,34.274,156.474
C09875=1043.838,-74.269,-73.979,169.350,34.275,156.475
C09876=1043.844,-74.019,-73.990,169.352,34.275,156.475
C09877=1043.850,-73.770,-74.002,169.354,34.276,156.475
C09878=1043.856,-73.520,-74.013,169.357,34.276,156.475
C09879=1043.863,-73.271,-74.025,169.359,34.277,156.475
C09880=1043.868,-73.021,-74.036,169.361,34.277,156.475
C09881=1043.875,-72.771,-74.048,169.363,34.278,156.475
C09882=1043.880,-72.522,-74.059,169.366,34.279,156.475
C09883=1043.887,-72.272,-74.071,169.368,34.280,156.475
C09884=1043.892,-72.022,-74.083,169.370,34.280,156.475
C09885=1043.899,-71.773,-74.095,169.372,34.280,156.475
C09886=1043.905,-71.523,-74.106,169.375,34.281,156.475
C09887=1043.911,-71.274,-74.117,169.377,34.282,156.475
C09888=1043.917,-71.023,-74.129,169.379,34.283,156.475
C09889=1043.923,-70.774,-74.141,169.381,34.284,156.475
C09890=1043.929,-70.524,-74.152,169.384,34.284,156.475
C09891=1043.936,-70.275,-74.164,169.386,34.285,156.475
C09892=1043.941,-70.025,-74.176,169.388,34.285,156.475
C09893=1043.947,-69.775,-74.187,169.390,34.286,156.476
C09894=1043.953,-69.526,-74.199,169.392,34.287,156.476
C09895=1043.960,-69.276,-74.210,169.395,34.287,156.476
C09896=1043.966,-69.026,-74.223,169.397,34.288,156.476
C09897=1043.971,-68.777,-74.234,169.399,34.288,156.476
C09898=1043.978,-68.527,-74.246,169.401,34.289,156.476
C09899=1043.985,-68.278,-74.258,169.404,34.290,156.476
C09900=1043.990,-68.028,-74.269,169.406,34.291,156.476
C09901=1043.997,-67.745,-74.283,169.408,34.292,156.476
C09902=1044.004,-67.462,-74.296,169.411,34.292,156.476
C09903=1044.011,-67.180,-74.309,169.413,34.293,156.476
C09904=1044.018,-66.898,-74.323,169.416,34.294,156.476
C09905=1044.024,-66.647,-74.334,169.418,34.294,156.476
C09906=1044.030,-66.399,-74.346,169.420,34.295,156.476
C09907=1044.037,-66.149,-74.358,169.423,34.296,156.476
C09908=1044.043,-65.898,-74.370,169.425,34.296,156.477
C09909=1044.049,-65.649,-74.382,169.427,34.297,156.477
C09910=1044.055,-65.400,-74.393,169.429,34.298,156.477
C09911=1044.061,-65.150,-74.406,169.431,34.299,156.477
C09912=1044.067,-64.900,-74.417,169.434,34.299,156.477
C09913=1044.074,-64.651,-74.429,169.436,34.300,156.477
C09914=1044.080,-64.402,-74.440,169.438,34.300,156.477
C09915=1044.086,-64.152,-74.453,169.440,34.301,156.477
C09916=1044.092,-63.901,-74.464,169.442,34.302,156.477
C09917=1044.098,-63.653,-74.476,169.445,34.303,156.477
C09918=1044.104,-63.403,-74.488,169.447,34.303,156.477
C09919=1044.111,-63.153,-74.500,169.449,34.304,156.477
C09920=1044.118,-62.904,-74.512,169.451,34.305,156.477
C09921=1044.123,-62.653,-74.524,169.454,34.306,156.477
C09922=1044.129,-62.404,-74.536,169.456,34.306,156.478
C09923=1044.136,-62.155,-74.548,169.458,34.307,156.478
C09924=1044.142,-61.905,-74.560,169.460,34.307,156.478
C09925=1044.149,-61.655,-74.572,169.462,34.308,156.478
C09926=1044.155,-61.406,-74.584,169.465,34.309,156.478
C09927=1044.160,-61.156,-74.596,169.467,34.310,156.478
C09928=1044.167,-60.906,-74.608,169.469,34.310,156.478
C09929=1044.173,-60.657,-74.620,169.472,34.311,156.478
C09930=1044.179,-60.407,-74.632,169.474,34.312,156.478
C09931=1044.186,-60.157,-74.644,169.477,34.313,156.478
C09932=1044.193,-59.908,-74.656,169.479,34.313,156.478
C09933=1044.198,-59.658,-74.668,169.481,34.314,156.478
C09934=1044.205,-59.409,-74.680,169.483,34.315,156.478
C09935=1044.211,-59.159,-74.692,169.485,34.316,156.479
C09936=1044.217,-58.909,-74.704,169.487,34.317,156.479
C09937=1044.224,-58.659,-74.716,169.490,34.317,156.479
C09938=1044.230,-58.410,-74.728,169.492,34.317,156.479
C09939=1044.236,-58.160,-74.740,169.494,34.318,156.479
C09940=1044.242,-57.911,-74.752,169.496,34.319,156.479
C09941=1044.249,-57.661,-74.764,169.498,34.320,156.479
C09942=1044.255,-57.411,-74.777,169.501,34.321,156.479
C09943=1044.261,-57.162,-74.789,169.503,34.321,156.479
C09944=1044.268,-56.912,-74.801,169.505,34.322,156.479
C09945=1044.278,-56.496,-74.821,169.509,34.324,156.479
C09946=1044.289,-56.080,-74.842,169.512,34.324,156.479
C09947=1044.300,-55.664,-74.861,169.516,34.326,156.480
C09948=1044.310,-55.248,-74.882,169.520,34.327,156.480
C09949=1044.317,-54.998,-74.894,169.522,34.328,156.480
C09950=1044.323,-54.748,-74.907,169.524,34.329,156.480
C09951=1044.329,-54.499,-74.919,169.526,34.330,156.480
C09952=1044.335,-54.249,-74.931,169.528,34.330,156.480
C09953=1044.342,-53.999,-74.943,169.530,34.331,156.480
C09954=1044.349,-53.750,-74.955,169.533,34.332,156.480
C09955=1044.355,-53.500,-74.968,169.535,34.333,156.480
C09956=1044.361,-53.251,-74.980,169.537,34.333,156.480
C09957=1044.367,-53.001,-74.993,169.539,34.334,156.480
C09958=1044.374,-52.751,-75.005,169.541,34.335,156.481
C09959=1044.381,-52.502,-75.017,169.543,34.336,156.481
C09960=1044.387,-52.252,-75.029,169.546,34.336,156.481
C09961=1044.395,-51.888,-75.047,169.549,34.337,156.481
C09962=1044.405,-51.523,-75.065,169.552,34.339,156.481
C09963=1044.414,-51.159,-75.083,169.555,34.340,156.481
C09964=1044.424,-50.795,-75.102,169.558,34.341,156.481
C09965=1044.430,-50.545,-75.114,169.560,34.342,156.481
C09966=1044.437,-50.296,-75.126,169.563,34.343,156.481
C09967=1044.443,-50.046,-75.139,169.565,34.343,156.482
C09968=1044.449,-49.796,-75.152,169.567,34.344,156.482
C09969=1044.455,-49.547,-75.164,169.569,34.345,156.482
C09970=1044.461,-49.297,-75.176,169.571,34.346,156.482
C09971=1044.467,-49.047,-75.189,169.573,34.347,156.482
C09972=1044.474,-48.798,-75.202,169.575,34.348,156.482
C09973=1044.480,-48.548,-75.215,169.577,34.349,156.482
C09974=1044.486,-48.298,-75.227,169.579,34.350,156.482
C09975=1044.492,-48.049,-75.240,169.582,34.351,156.482
C09976=1044.498,-47.799,-75.253,169.584,34.352,156.483
C09977=1044.504,-47.549,-75.265,169.586,34.353,156.483
C09978=1044.511,-47.300,-75.278,169.588,34.354,156.483
C09979=1044.517,-47.050,-75.290,169.590,34.354,156.483
C09980=1044.523,-46.801,-75.304,169.592,34.356,156.483
C09981=1044.529,-46.551,-75.316,169.594,34.356,156.483
C09982=1044.536,-46.302,-75.328,169.596,34.357,156.483
C09983=1044.542,-46.052,-75.341,169.598,34.358,156.483
C09984=1044.548,-45.803,-75.354,169.601,34.359,156.484
C09985=1044.554,-45.553,-75.367,169.603,34.360,156.484
C09986=1044.561,-45.304,-75.379,169.605,34.361,156.484
C09987=1044.568,-45.054,-75.393,169.607,34.362,156.484
C09988=1044.574,-44.804,-75.405,169.609,34.363,156.484
C09989=1044.579,-44.554,-75.418,169.611,34.364,156.484
C09990=1044.586,-44.305,-75.431,169.613,34.364,156.484
C09991=1044.592,-44.055,-75.443,169.615,34.366,156.484
C09992=1044.599,-43.806,-75.456,169.617,34.367,156.484
C09993=1044.604,-43.556,-75.469,169.619,34.367,156.485
C09994=1044.611,-43.307,-75.482,169.622,34.369,156.485
C09995=1044.617,-43.057,-75.495,169.624,34.370,156.485
C09996=1044.624,-42.808,-75.507,169.626,34.370,156.485
//INST
///DATE 2021/06/17 10:56
///ATTR SC,RW,RJ
////FRAME ROBOT
///GROUP1 RB1
NOP
MOVL C00000 V=800.0 PL=0
MOVL C00001 V=800.0 PL=0
MOVL C00002 V=800.0 PL=0
MOVL C00003 V=800.0 PL=0
MOVL C00004 V=800.0 PL=0
MOVL C00005 V=800.0 PL=0
MOVL C00006 V=800.0 PL=0
MOVL C00007 V=800.0 PL=0
MOVL C00008 V=800.0 PL=0
MOVL C00009 V=800.0 PL=0
MOVL C00010 V=800.0 PL=0
MOVL C00011 V=800.0 PL=0
MOVL C00012 V=800.0 PL=0
MOVL C00013 V=800.0 PL=0
MOVL C00014 V=800.0 PL=0
MOVL C00015 V=800.0 PL=0
MOVL C00016 V=800.0 PL=0
MOVL C00017 V=800.0 PL=0
MOVL C00018 V=800.0 PL=0
MOVL C00019 V=800.0 PL=0
MOVL C00020 V=800.0 PL=0
MOVL C00021 V=800.0 PL=0
MOVL C00022 V=800.0 PL=0
MOVL C00023 V=800.0 PL=0
MOVL C00024 V=800.0 PL=0
MOVL C00025 V=800.0 PL=0
MOVL C00026 V=800.0 PL=0
MOVL C00027 V=800.0 PL=0
MOVL C00028 V=800.0 PL=0
MOVL C00029 V=800.0 PL=0
MOVL C00030 V=800.0 PL=0
MOVL C00031 V=800.0 PL=0
MOVL C00032 V=800.0 PL=0
MOVL C00033 V=800.0 PL=0
MOVL C00034 V=800.0 PL=0
MOVL C00035 V=800.0 PL=0
MOVL C00036 V=800.0 PL=0
MOVL C00037 V=800.0 PL=0
MOVL C00038 V=800.0 PL=0
MOVL C00039 V=800.0 PL=0
MOVL C00040 V=800.0 PL=0
MOVL C00041 V=800.0 PL=0
MOVL C00042 V=800.0 PL=0
MOVL C00043 V=800.0 PL=0
MOVL C00044 V=800.0 PL=0
MOVL C00045 V=800.0 PL=0
MOVL C00046 V=800.0 PL=0
MOVL C00047 V=800.0 PL=0
MOVL C00048 V=800.0 PL=0
MOVL C00049 V=800.0 PL=0
MOVL C00050 V=800.0 PL=0
MOVL C00051 V=800.0 PL=0
MOVL C00052 V=800.0 PL=0
MOVL C00053 V=800.0 PL=0
MOVL C00054 V=800.0 PL=0
MOVL C00055 V=800.0 PL=0
MOVL C00056 V=800.0 PL=0
MOVL C00057 V=800.0 PL=0
MOVL C00058 V=800.0 PL=0
MOVL C00059 V=800.0 PL=0
MOVL C00060 V=800.0 PL=0
MOVL C00061 V=800.0 PL=0
MOVL C00062 V=800.0 PL=0
MOVL C00063 V=800.0 PL=0
MOVL C00064 V=800.0 PL=0
MOVL C00065 V=800.0 PL=0
MOVL C00066 V=800.0 PL=0
MOVL C00067 V=800.0 PL=0
MOVL C00068 V=800.0 PL=0
MOVL C00069 V=800.0 PL=0
MOVL C00070 V=800.0 PL=0
MOVL C00071 V=800.0 PL=0
MOVL C00072 V=800.0 PL=0
MOVL C00073 V=800.0 PL=0
MOVL C00074 V=800.0 PL=0
MOVL C00075 V=800.0 PL=0
MOVL C00076 V=800.0 PL=0
MOVL C00077 V=800.0 PL=0
MOVL C00078 V=800.0 PL=0
MOVL C00079 V=800.0 PL=0
MOVL C00080 V=800.0 PL=0
MOVL C00081 V=800.0 PL=0
MOVL C00082 V=800.0 PL=0
MOVL C00083 V=800.0 PL=0
MOVL C00084 V=800.0 PL=0
MOVL C00085 V=800.0 PL=0
MOVL C00086 V=800.0 PL=0
MOVL C00087 V=800.0 PL=0
MOVL C00088 V=800.0 PL=0
MOVL C00089 V=800.0 PL=0
MOVL C00090 V=800.0 PL=0
MOVL C00091 V=800.0 PL=0
MOVL C00092 V=800.0 PL=0
MOVL C00093 V=800.0 PL=0
MOVL C00094 V=800.0 PL=0
MOVL C00095 V=800.0 PL=0
MOVL C00096 V=800.0 PL=0
MOVL C00097 V=800.0 PL=0
MOVL C00098 V=800.0 PL=0
MOVL C00099 V=800.0 PL=0
MOVL C00100 V=800.0 PL=0
MOVL C00101 V=800.0 PL=0
MOVL C00102 V=800.0 PL=0
MOVL C00103 V=800.0 PL=0
MOVL C00104 V=800.0 PL=0
MOVL C00105 V=800.0 PL=0
MOVL C00106 V=800.0 PL=0
MOVL C00107 V=800.0 PL=0
MOVL C00108 V=800.0 PL=0
MOVL C00109 V=800.0 PL=0
MOVL C00110 V=800.0 PL=0
MOVL C00111 V=800.0 PL=0
MOVL C00112 V=800.0 PL=0
MOVL C00113 V=800.0 PL=0
MOVL C00114 V=800.0 PL=0
MOVL C00115 V=800.0 PL=0
MOVL C00116 V=800.0 PL=0
MOVL C00117 V=800.0 PL=0
MOVL C00118 V=800.0 PL=0
MOVL C00119 V=800.0 PL=0
MOVL C00120 V=800.0 PL=0
MOVL C00121 V=800.0 PL=0
MOVL C00122 V=800.0 PL=0
MOVL C00123 V=800.0 PL=0
MOVL C00124 V=800.0 PL=0
MOVL C00125 V=800.0 PL=0
MOVL C00126 V=800.0 PL=0
MOVL C00127 V=800.0 PL=0
MOVL C00128 V=800.0 PL=0
MOVL C00129 V=800.0 PL=0
MOVL C00130 V=800.0 PL=0
MOVL C00131 V=800.0 PL=0
MOVL C00132 V=800.0 PL=0
MOVL C00133 V=800.0 PL=0
MOVL C00134 V=800.0 PL=0
MOVL C00135 V=800.0 PL=0
MOVL C00136 V=800.0 PL=0
MOVL C00137 V=800.0 PL=0
MOVL C00138 V=800.0 PL=0
MOVL C00139 V=800.0 PL=0
MOVL C00140 V=800.0 PL=0
MOVL C00141 V=800.0 PL=0
MOVL C00142 V=800.0 PL=0
MOVL C00143 V=800.0 PL=0
MOVL C00144 V=800.0 PL=0
MOVL C00145 V=800.0 PL=0
MOVL C00146 V=800.0 PL=0
MOVL C00147 V=800.0 PL=0
MOVL C00148 V=800.0 PL=0
MOVL C00149 V=800.0 PL=0
MOVL C00150 V=800.0 PL=0
MOVL C00151 V=800.0 PL=0
MOVL C00152 V=800.0 PL=0
MOVL C00153 V=800.0 PL=0
MOVL C00154 V=800.0 PL=0
MOVL C00155 V=800.0 PL=0
MOVL C00156 V=800.0 PL=0
MOVL C00157 V=800.0 PL=0
MOVL C00158 V=800.0 PL=0
MOVL C00159 V=800.0 PL=0
MOVL C00160 V=800.0 PL=0
MOVL C00161 V=800.0 PL=0
MOVL C00162 V=800.0 PL=0
MOVL C00163 V=800.0 PL=0
MOVL C00164 V=800.0 PL=0
MOVL C00165 V=800.0 PL=0
MOVL C00166 V=800.0 PL=0
MOVL C00167 V=800.0 PL=0
MOVL C00168 V=800.0 PL=0
MOVL C00169 V=800.0 PL=0
MOVL C00170 V=800.0 PL=0
MOVL C00171 V=800.0 PL=0
MOVL C00172 V=800.0 PL=0
MOVL C00173 V=800.0 PL=0
MOVL C00174 V=800.0 PL=0
MOVL C00175 V=800.0 PL=0
MOVL C00176 V=800.0 PL=0
MOVL C00177 V=800.0 PL=0
MOVL C00178 V=800.0 PL=0
MOVL C00179 V=800.0 PL=0
MOVL C00180 V=800.0 PL=0
MOVL C00181 V=800.0 PL=0
MOVL C00182 V=800.0 PL=0
MOVL C00183 V=800.0 PL=0
MOVL C00184 V=800.0 PL=0
MOVL C00185 V=800.0 PL=0
MOVL C00186 V=800.0 PL=0
MOVL C00187 V=800.0 PL=0
MOVL C00188 V=800.0 PL=0
MOVL C00189 V=800.0 PL=0
MOVL C00190 V=800.0 PL=0
MOVL C00191 V=800.0 PL=0
MOVL C00192 V=800.0 PL=0
MOVL C00193 V=800.0 PL=0
MOVL C00194 V=800.0 PL=0
MOVL C00195 V=800.0 PL=0
MOVL C00196 V=800.0 PL=0
MOVL C00197 V=800.0 PL=0
MOVL C00198 V=800.0 PL=0
MOVL C00199 V=800.0 PL=0
MOVL C00200 V=800.0 PL=0
MOVL C00201 V=800.0 PL=0
MOVL C00202 V=800.0 PL=0
MOVL C00203 V=800.0 PL=0
MOVL C00204 V=800.0 PL=0
MOVL C00205 V=800.0 PL=0
MOVL C00206 V=800.0 PL=0
MOVL C00207 V=800.0 PL=0
MOVL C00208 V=800.0 PL=0
MOVL C00209 V=800.0 PL=0
MOVL C00210 V=800.0 PL=0
MOVL C00211 V=800.0 PL=0
MOVL C00212 V=800.0 PL=0
MOVL C00213 V=800.0 PL=0
MOVL C00214 V=800.0 PL=0
MOVL C00215 V=800.0 PL=0
MOVL C00216 V=800.0 PL=0
MOVL C00217 V=800.0 PL=0
MOVL C00218 V=800.0 PL=0
MOVL C00219 V=800.0 PL=0
MOVL C00220 V=800.0 PL=0
MOVL C00221 V=800.0 PL=0
MOVL C00222 V=800.0 PL=0
MOVL C00223 V=800.0 PL=0
MOVL C00224 V=800.0 PL=0
MOVL C00225 V=800.0 PL=0
MOVL C00226 V=800.0 PL=0
MOVL C00227 V=800.0 PL=0
MOVL C00228 V=800.0 PL=0
MOVL C00229 V=800.0 PL=0
MOVL C00230 V=800.0 PL=0
MOVL C00231 V=800.0 PL=0
MOVL C00232 V=800.0 PL=0
MOVL C00233 V=800.0 PL=0
MOVL C00234 V=800.0 PL=0
MOVL C00235 V=800.0 PL=0
MOVL C00236 V=800.0 PL=0
MOVL C00237 V=800.0 PL=0
MOVL C00238 V=800.0 PL=0
MOVL C00239 V=800.0 PL=0
MOVL C00240 V=800.0 PL=0
MOVL C00241 V=800.0 PL=0
MOVL C00242 V=800.0 PL=0
MOVL C00243 V=800.0 PL=0
MOVL C00244 V=800.0 PL=0
MOVL C00245 V=800.0 PL=0
MOVL C00246 V=800.0 PL=0
MOVL C00247 V=800.0 PL=0
MOVL C00248 V=800.0 PL=0
MOVL C00249 V=800.0 PL=0
MOVL C00250 V=800.0 PL=0
MOVL C00251 V=800.0 PL=0
MOVL C00252 V=800.0 PL=0
MOVL C00253 V=800.0 PL=0
MOVL C00254 V=800.0 PL=0
MOVL C00255 V=800.0 PL=0
MOVL C00256 V=800.0 PL=0
MOVL C00257 V=800.0 PL=0
MOVL C00258 V=800.0 PL=0
MOVL C00259 V=800.0 PL=0
MOVL C00260 V=800.0 PL=0
MOVL C00261 V=800.0 PL=0
MOVL C00262 V=800.0 PL=0
MOVL C00263 V=800.0 PL=0
MOVL C00264 V=800.0 PL=0
MOVL C00265 V=800.0 PL=0
MOVL C00266 V=800.0 PL=0
MOVL C00267 V=800.0 PL=0
MOVL C00268 V=800.0 PL=0
MOVL C00269 V=800.0 PL=0
MOVL C00270 V=800.0 PL=0
MOVL C00271 V=800.0 PL=0
MOVL C00272 V=800.0 PL=0
MOVL C00273 V=800.0 PL=0
MOVL C00274 V=800.0 PL=0
MOVL C00275 V=800.0 PL=0
MOVL C00276 V=800.0 PL=0
MOVL C00277 V=800.0 PL=0
MOVL C00278 V=800.0 PL=0
MOVL C00279 V=800.0 PL=0
MOVL C00280 V=800.0 PL=0
MOVL C00281 V=800.0 PL=0
MOVL C00282 V=800.0 PL=0
MOVL C00283 V=800.0 PL=0
MOVL C00284 V=800.0 PL=0
MOVL C00285 V=800.0 PL=0
MOVL C00286 V=800.0 PL=0
MOVL C00287 V=800.0 PL=0
MOVL C00288 V=800.0 PL=0
MOVL C00289 V=800.0 PL=0
MOVL C00290 V=800.0 PL=0
MOVL C00291 V=800.0 PL=0
MOVL C00292 V=800.0 PL=0
MOVL C00293 V=800.0 PL=0
MOVL C00294 V=800.0 PL=0
MOVL C00295 V=800.0 PL=0
MOVL C00296 V=800.0 PL=0
MOVL C00297 V=800.0 PL=0
MOVL C00298 V=800.0 PL=0
MOVL C00299 V=800.0 PL=0
MOVL C00300 V=800.0 PL=0
MOVL C00301 V=800.0 PL=0
MOVL C00302 V=800.0 PL=0
MOVL C00303 V=800.0 PL=0
MOVL C00304 V=800.0 PL=0
MOVL C00305 V=800.0 PL=0
MOVL C00306 V=800.0 PL=0
MOVL C00307 V=800.0 PL=0
MOVL C00308 V=800.0 PL=0
MOVL C00309 V=800.0 PL=0
MOVL C00310 V=800.0 PL=0
MOVL C00311 V=800.0 PL=0
MOVL C00312 V=800.0 PL=0
MOVL C00313 V=800.0 PL=0
MOVL C00314 V=800.0 PL=0
MOVL C00315 V=800.0 PL=0
MOVL C00316 V=800.0 PL=0
MOVL C00317 V=800.0 PL=0
MOVL C00318 V=800.0 PL=0
MOVL C00319 V=800.0 PL=0
MOVL C00320 V=800.0 PL=0
MOVL C00321 V=800.0 PL=0
MOVL C00322 V=800.0 PL=0
MOVL C00323 V=800.0 PL=0
MOVL C00324 V=800.0 PL=0
MOVL C00325 V=800.0 PL=0
MOVL C00326 V=800.0 PL=0
MOVL C00327 V=800.0 PL=0
MOVL C00328 V=800.0 PL=0
MOVL C00329 V=800.0 PL=0
MOVL C00330 V=800.0 PL=0
MOVL C00331 V=800.0 PL=0
MOVL C00332 V=800.0 PL=0
MOVL C00333 V=800.0 PL=0
MOVL C00334 V=800.0 PL=0
MOVL C00335 V=800.0 PL=0
MOVL C00336 V=800.0 PL=0
MOVL C00337 V=800.0 PL=0
MOVL C00338 V=800.0 PL=0
MOVL C00339 V=800.0 PL=0
MOVL C00340 V=800.0 PL=0
MOVL C00341 V=800.0 PL=0
MOVL C00342 V=800.0 PL=0
MOVL C00343 V=800.0 PL=0
MOVL C00344 V=800.0 PL=0
MOVL C00345 V=800.0 PL=0
MOVL C00346 V=800.0 PL=0
MOVL C00347 V=800.0 PL=0
MOVL C00348 V=800.0 PL=0
MOVL C00349 V=800.0 PL=0
MOVL C00350 V=800.0 PL=0
MOVL C00351 V=800.0 PL=0
MOVL C00352 V=800.0 PL=0
MOVL C00353 V=800.0 PL=0
MOVL C00354 V=800.0 PL=0
MOVL C00355 V=800.0 PL=0
MOVL C00356 V=800.0 PL=0
MOVL C00357 V=800.0 PL=0
MOVL C00358 V=800.0 PL=0
MOVL C00359 V=800.0 PL=0
MOVL C00360 V=800.0 PL=0
MOVL C00361 V=800.0 PL=0
MOVL C00362 V=800.0 PL=0
MOVL C00363 V=800.0 PL=0
MOVL C00364 V=800.0 PL=0
MOVL C00365 V=800.0 PL=0
MOVL C00366 V=800.0 PL=0
MOVL C00367 V=800.0 PL=0
MOVL C00368 V=800.0 PL=0
MOVL C00369 V=800.0 PL=0
MOVL C00370 V=800.0 PL=0
MOVL C00371 V=800.0 PL=0
MOVL C00372 V=800.0 PL=0
MOVL C00373 V=800.0 PL=0
MOVL C00374 V=800.0 PL=0
MOVL C00375 V=800.0 PL=0
MOVL C00376 V=800.0 PL=0
MOVL C00377 V=800.0 PL=0
MOVL C00378 V=800.0 PL=0
MOVL C00379 V=800.0 PL=0
MOVL C00380 V=800.0 PL=0
MOVL C00381 V=800.0 PL=0
MOVL C00382 V=800.0 PL=0
MOVL C00383 V=800.0 PL=0
MOVL C00384 V=800.0 PL=0
MOVL C00385 V=800.0 PL=0
MOVL C00386 V=800.0 PL=0
MOVL C00387 V=800.0 PL=0
MOVL C00388 V=800.0 PL=0
MOVL C00389 V=800.0 PL=0
MOVL C00390 V=800.0 PL=0
MOVL C00391 V=800.0 PL=0
MOVL C00392 V=800.0 PL=0
MOVL C00393 V=800.0 PL=0
MOVL C00394 V=800.0 PL=0
MOVL C00395 V=800.0 PL=0
MOVL C00396 V=800.0 PL=0
MOVL C00397 V=800.0 PL=0
MOVL C00398 V=800.0 PL=0
MOVL C00399 V=800.0 PL=0
MOVL C00400 V=800.0 PL=0
MOVL C00401 V=800.0 PL=0
MOVL C00402 V=800.0 PL=0
MOVL C00403 V=800.0 PL=0
MOVL C00404 V=800.0 PL=0
MOVL C00405 V=800.0 PL=0
MOVL C00406 V=800.0 PL=0
MOVL C00407 V=800.0 PL=0
MOVL C00408 V=800.0 PL=0
MOVL C00409 V=800.0 PL=0
MOVL C00410 V=800.0 PL=0
MOVL C00411 V=800.0 PL=0
MOVL C00412 V=800.0 PL=0
MOVL C00413 V=800.0 PL=0
MOVL C00414 V=800.0 PL=0
MOVL C00415 V=800.0 PL=0
MOVL C00416 V=800.0 PL=0
MOVL C00417 V=800.0 PL=0
MOVL C00418 V=800.0 PL=0
MOVL C00419 V=800.0 PL=0
MOVL C00420 V=800.0 PL=0
MOVL C00421 V=800.0 PL=0
MOVL C00422 V=800.0 PL=0
MOVL C00423 V=800.0 PL=0
MOVL C00424 V=800.0 PL=0
MOVL C00425 V=800.0 PL=0
MOVL C00426 V=800.0 PL=0
MOVL C00427 V=800.0 PL=0
MOVL C00428 V=800.0 PL=0
MOVL C00429 V=800.0 PL=0
MOVL C00430 V=800.0 PL=0
MOVL C00431 V=800.0 PL=0
MOVL C00432 V=800.0 PL=0
MOVL C00433 V=800.0 PL=0
MOVL C00434 V=800.0 PL=0
MOVL C00435 V=800.0 PL=0
MOVL C00436 V=800.0 PL=0
MOVL C00437 V=800.0 PL=0
MOVL C00438 V=800.0 PL=0
MOVL C00439 V=800.0 PL=0
MOVL C00440 V=800.0 PL=0
MOVL C00441 V=800.0 PL=0
MOVL C00442 V=800.0 PL=0
MOVL C00443 V=800.0 PL=0
MOVL C00444 V=800.0 PL=0
MOVL C00445 V=800.0 PL=0
MOVL C00446 V=800.0 PL=0
MOVL C00447 V=800.0 PL=0
MOVL C00448 V=800.0 PL=0
MOVL C00449 V=800.0 PL=0
MOVL C00450 V=800.0 PL=0
MOVL C00451 V=800.0 PL=0
MOVL C00452 V=800.0 PL=0
MOVL C00453 V=800.0 PL=0
MOVL C00454 V=800.0 PL=0
MOVL C00455 V=800.0 PL=0
MOVL C00456 V=800.0 PL=0
MOVL C00457 V=800.0 PL=0
MOVL C00458 V=800.0 PL=0
MOVL C00459 V=800.0 PL=0
MOVL C00460 V=800.0 PL=0
MOVL C00461 V=800.0 PL=0
MOVL C00462 V=800.0 PL=0
MOVL C00463 V=800.0 PL=0
MOVL C00464 V=800.0 PL=0
MOVL C00465 V=800.0 PL=0
MOVL C00466 V=800.0 PL=0
MOVL C00467 V=800.0 PL=0
MOVL C00468 V=800.0 PL=0
MOVL C00469 V=800.0 PL=0
MOVL C00470 V=800.0 PL=0
MOVL C00471 V=800.0 PL=0
MOVL C00472 V=800.0 PL=0
MOVL C00473 V=800.0 PL=0
MOVL C00474 V=800.0 PL=0
MOVL C00475 V=800.0 PL=0
MOVL C00476 V=800.0 PL=0
MOVL C00477 V=800.0 PL=0
MOVL C00478 V=800.0 PL=0
MOVL C00479 V=800.0 PL=0
MOVL C00480 V=800.0 PL=0
MOVL C00481 V=800.0 PL=0
MOVL C00482 V=800.0 PL=0
MOVL C00483 V=800.0 PL=0
MOVL C00484 V=800.0 PL=0
MOVL C00485 V=800.0 PL=0
MOVL C00486 V=800.0 PL=0
MOVL C00487 V=800.0 PL=0
MOVL C00488 V=800.0 PL=0
MOVL C00489 V=800.0 PL=0
MOVL C00490 V=800.0 PL=0
MOVL C00491 V=800.0 PL=0
MOVL C00492 V=800.0 PL=0
MOVL C00493 V=800.0 PL=0
MOVL C00494 V=800.0 PL=0
MOVL C00495 V=800.0 PL=0
MOVL C00496 V=800.0 PL=0
MOVL C00497 V=800.0 PL=0
MOVL C00498 V=800.0 PL=0
MOVL C00499 V=800.0 PL=0
MOVL C00500 V=800.0 PL=0
MOVL C00501 V=800.0 PL=0
MOVL C00502 V=800.0 PL=0
MOVL C00503 V=800.0 PL=0
MOVL C00504 V=800.0 PL=0
MOVL C00505 V=800.0 PL=0
MOVL C00506 V=800.0 PL=0
MOVL C00507 V=800.0 PL=0
MOVL C00508 V=800.0 PL=0
MOVL C00509 V=800.0 PL=0
MOVL C00510 V=800.0 PL=0
MOVL C00511 V=800.0 PL=0
MOVL C00512 V=800.0 PL=0
MOVL C00513 V=800.0 PL=0
MOVL C00514 V=800.0 PL=0
MOVL C00515 V=800.0 PL=0
MOVL C00516 V=800.0 PL=0
MOVL C00517 V=800.0 PL=0
MOVL C00518 V=800.0 PL=0
MOVL C00519 V=800.0 PL=0
MOVL C00520 V=800.0 PL=0
MOVL C00521 V=800.0 PL=0
MOVL C00522 V=800.0 PL=0
MOVL C00523 V=800.0 PL=0
MOVL C00524 V=800.0 PL=0
MOVL C00525 V=800.0 PL=0
MOVL C00526 V=800.0 PL=0
MOVL C00527 V=800.0 PL=0
MOVL C00528 V=800.0 PL=0
MOVL C00529 V=800.0 PL=0
MOVL C00530 V=800.0 PL=0
MOVL C00531 V=800.0 PL=0
MOVL C00532 V=800.0 PL=0
MOVL C00533 V=800.0 PL=0
MOVL C00534 V=800.0 PL=0
MOVL C00535 V=800.0 PL=0
MOVL C00536 V=800.0 PL=0
MOVL C00537 V=800.0 PL=0
MOVL C00538 V=800.0 PL=0
MOVL C00539 V=800.0 PL=0
MOVL C00540 V=800.0 PL=0
MOVL C00541 V=800.0 PL=0
MOVL C00542 V=800.0 PL=0
MOVL C00543 V=800.0 PL=0
MOVL C00544 V=800.0 PL=0
MOVL C00545 V=800.0 PL=0
MOVL C00546 V=800.0 PL=0
MOVL C00547 V=800.0 PL=0
MOVL C00548 V=800.0 PL=0
MOVL C00549 V=800.0 PL=0
MOVL C00550 V=800.0 PL=0
MOVL C00551 V=800.0 PL=0
MOVL C00552 V=800.0 PL=0
MOVL C00553 V=800.0 PL=0
MOVL C00554 V=800.0 PL=0
MOVL C00555 V=800.0 PL=0
MOVL C00556 V=800.0 PL=0
MOVL C00557 V=800.0 PL=0
MOVL C00558 V=800.0 PL=0
MOVL C00559 V=800.0 PL=0
MOVL C00560 V=800.0 PL=0
MOVL C00561 V=800.0 PL=0
MOVL C00562 V=800.0 PL=0
MOVL C00563 V=800.0 PL=0
MOVL C00564 V=800.0 PL=0
MOVL C00565 V=800.0 PL=0
MOVL C00566 V=800.0 PL=0
MOVL C00567 V=800.0 PL=0
MOVL C00568 V=800.0 PL=0
MOVL C00569 V=800.0 PL=0
MOVL C00570 V=800.0 PL=0
MOVL C00571 V=800.0 PL=0
MOVL C00572 V=800.0 PL=0
MOVL C00573 V=800.0 PL=0
MOVL C00574 V=800.0 PL=0
MOVL C00575 V=800.0 PL=0
MOVL C00576 V=800.0 PL=0
MOVL C00577 V=800.0 PL=0
MOVL C00578 V=800.0 PL=0
MOVL C00579 V=800.0 PL=0
MOVL C00580 V=800.0 PL=0
MOVL C00581 V=800.0 PL=0
MOVL C00582 V=800.0 PL=0
MOVL C00583 V=800.0 PL=0
MOVL C00584 V=800.0 PL=0
MOVL C00585 V=800.0 PL=0
MOVL C00586 V=800.0 PL=0
MOVL C00587 V=800.0 PL=0
MOVL C00588 V=800.0 PL=0
MOVL C00589 V=800.0 PL=0
MOVL C00590 V=800.0 PL=0
MOVL C00591 V=800.0 PL=0
MOVL C00592 V=800.0 PL=0
MOVL C00593 V=800.0 PL=0
MOVL C00594 V=800.0 PL=0
MOVL C00595 V=800.0 PL=0
MOVL C00596 V=800.0 PL=0
MOVL C00597 V=800.0 PL=0
MOVL C00598 V=800.0 PL=0
MOVL C00599 V=800.0 PL=0
MOVL C00600 V=800.0 PL=0
MOVL C00601 V=800.0 PL=0
MOVL C00602 V=800.0 PL=0
MOVL C00603 V=800.0 PL=0
MOVL C00604 V=800.0 PL=0
MOVL C00605 V=800.0 PL=0
MOVL C00606 V=800.0 PL=0
MOVL C00607 V=800.0 PL=0
MOVL C00608 V=800.0 PL=0
MOVL C00609 V=800.0 PL=0
MOVL C00610 V=800.0 PL=0
MOVL C00611 V=800.0 PL=0
MOVL C00612 V=800.0 PL=0
MOVL C00613 V=800.0 PL=0
MOVL C00614 V=800.0 PL=0
MOVL C00615 V=800.0 PL=0
MOVL C00616 V=800.0 PL=0
MOVL C00617 V=800.0 PL=0
MOVL C00618 V=800.0 PL=0
MOVL C00619 V=800.0 PL=0
MOVL C00620 V=800.0 PL=0
MOVL C00621 V=800.0 PL=0
MOVL C00622 V=800.0 PL=0
MOVL C00623 V=800.0 PL=0
MOVL C00624 V=800.0 PL=0
MOVL C00625 V=800.0 PL=0
MOVL C00626 V=800.0 PL=0
MOVL C00627 V=800.0 PL=0
MOVL C00628 V=800.0 PL=0
MOVL C00629 V=800.0 PL=0
MOVL C00630 V=800.0 PL=0
MOVL C00631 V=800.0 PL=0
MOVL C00632 V=800.0 PL=0
MOVL C00633 V=800.0 PL=0
MOVL C00634 V=800.0 PL=0
MOVL C00635 V=800.0 PL=0
MOVL C00636 V=800.0 PL=0
MOVL C00637 V=800.0 PL=0
MOVL C00638 V=800.0 PL=0
MOVL C00639 V=800.0 PL=0
MOVL C00640 V=800.0 PL=0
MOVL C00641 V=800.0 PL=0
MOVL C00642 V=800.0 PL=0
MOVL C00643 V=800.0 PL=0
MOVL C00644 V=800.0 PL=0
MOVL C00645 V=800.0 PL=0
MOVL C00646 V=800.0 PL=0
MOVL C00647 V=800.0 PL=0
MOVL C00648 V=800.0 PL=0
MOVL C00649 V=800.0 PL=0
MOVL C00650 V=800.0 PL=0
MOVL C00651 V=800.0 PL=0
MOVL C00652 V=800.0 PL=0
MOVL C00653 V=800.0 PL=0
MOVL C00654 V=800.0 PL=0
MOVL C00655 V=800.0 PL=0
MOVL C00656 V=800.0 PL=0
MOVL C00657 V=800.0 PL=0
MOVL C00658 V=800.0 PL=0
MOVL C00659 V=800.0 PL=0
MOVL C00660 V=800.0 PL=0
MOVL C00661 V=800.0 PL=0
MOVL C00662 V=800.0 PL=0
MOVL C00663 V=800.0 PL=0
MOVL C00664 V=800.0 PL=0
MOVL C00665 V=800.0 PL=0
MOVL C00666 V=800.0 PL=0
MOVL C00667 V=800.0 PL=0
MOVL C00668 V=800.0 PL=0
MOVL C00669 V=800.0 PL=0
MOVL C00670 V=800.0 PL=0
MOVL C00671 V=800.0 PL=0
MOVL C00672 V=800.0 PL=0
MOVL C00673 V=800.0 PL=0
MOVL C00674 V=800.0 PL=0
MOVL C00675 V=800.0 PL=0
MOVL C00676 V=800.0 PL=0
MOVL C00677 V=800.0 PL=0
MOVL C00678 V=800.0 PL=0
MOVL C00679 V=800.0 PL=0
MOVL C00680 V=800.0 PL=0
MOVL C00681 V=800.0 PL=0
MOVL C00682 V=800.0 PL=0
MOVL C00683 V=800.0 PL=0
MOVL C00684 V=800.0 PL=0
MOVL C00685 V=800.0 PL=0
MOVL C00686 V=800.0 PL=0
MOVL C00687 V=800.0 PL=0
MOVL C00688 V=800.0 PL=0
MOVL C00689 V=800.0 PL=0
MOVL C00690 V=800.0 PL=0
MOVL C00691 V=800.0 PL=0
MOVL C00692 V=800.0 PL=0
MOVL C00693 V=800.0 PL=0
MOVL C00694 V=800.0 PL=0
MOVL C00695 V=800.0 PL=0
MOVL C00696 V=800.0 PL=0
MOVL C00697 V=800.0 PL=0
MOVL C00698 V=800.0 PL=0
MOVL C00699 V=800.0 PL=0
MOVL C00700 V=800.0 PL=0
MOVL C00701 V=800.0 PL=0
MOVL C00702 V=800.0 PL=0
MOVL C00703 V=800.0 PL=0
MOVL C00704 V=800.0 PL=0
MOVL C00705 V=800.0 PL=0
MOVL C00706 V=800.0 PL=0
MOVL C00707 V=800.0 PL=0
MOVL C00708 V=800.0 PL=0
MOVL C00709 V=800.0 PL=0
MOVL C00710 V=800.0 PL=0
MOVL C00711 V=800.0 PL=0
MOVL C00712 V=800.0 PL=0
MOVL C00713 V=800.0 PL=0
MOVL C00714 V=800.0 PL=0
MOVL C00715 V=800.0 PL=0
MOVL C00716 V=800.0 PL=0
MOVL C00717 V=800.0 PL=0
MOVL C00718 V=800.0 PL=0
MOVL C00719 V=800.0 PL=0
MOVL C00720 V=800.0 PL=0
MOVL C00721 V=800.0 PL=0
MOVL C00722 V=800.0 PL=0
MOVL C00723 V=800.0 PL=0
MOVL C00724 V=800.0 PL=0
MOVL C00725 V=800.0 PL=0
MOVL C00726 V=800.0 PL=0
MOVL C00727 V=800.0 PL=0
MOVL C00728 V=800.0 PL=0
MOVL C00729 V=800.0 PL=0
MOVL C00730 V=800.0 PL=0
MOVL C00731 V=800.0 PL=0
MOVL C00732 V=800.0 PL=0
MOVL C00733 V=800.0 PL=0
MOVL C00734 V=800.0 PL=0
MOVL C00735 V=800.0 PL=0
MOVL C00736 V=800.0 PL=0
MOVL C00737 V=800.0 PL=0
MOVL C00738 V=800.0 PL=0
MOVL C00739 V=800.0 PL=0
MOVL C00740 V=800.0 PL=0
MOVL C00741 V=800.0 PL=0
MOVL C00742 V=800.0 PL=0
MOVL C00743 V=800.0 PL=0
MOVL C00744 V=800.0 PL=0
MOVL C00745 V=800.0 PL=0
MOVL C00746 V=800.0 PL=0
MOVL C00747 V=800.0 PL=0
MOVL C00748 V=800.0 PL=0
MOVL C00749 V=800.0 PL=0
MOVL C00750 V=800.0 PL=0
MOVL C00751 V=800.0 PL=0
MOVL C00752 V=800.0 PL=0
MOVL C00753 V=800.0 PL=0
MOVL C00754 V=800.0 PL=0
MOVL C00755 V=800.0 PL=0
MOVL C00756 V=800.0 PL=0
MOVL C00757 V=800.0 PL=0
MOVL C00758 V=800.0 PL=0
MOVL C00759 V=800.0 PL=0
MOVL C00760 V=800.0 PL=0
MOVL C00761 V=800.0 PL=0
MOVL C00762 V=800.0 PL=0
MOVL C00763 V=800.0 PL=0
MOVL C00764 V=800.0 PL=0
MOVL C00765 V=800.0 PL=0
MOVL C00766 V=800.0 PL=0
MOVL C00767 V=800.0 PL=0
MOVL C00768 V=800.0 PL=0
MOVL C00769 V=800.0 PL=0
MOVL C00770 V=800.0 PL=0
MOVL C00771 V=800.0 PL=0
MOVL C00772 V=800.0 PL=0
MOVL C00773 V=800.0 PL=0
MOVL C00774 V=800.0 PL=0
MOVL C00775 V=800.0 PL=0
MOVL C00776 V=800.0 PL=0
MOVL C00777 V=800.0 PL=0
MOVL C00778 V=800.0 PL=0
MOVL C00779 V=800.0 PL=0
MOVL C00780 V=800.0 PL=0
MOVL C00781 V=800.0 PL=0
MOVL C00782 V=800.0 PL=0
MOVL C00783 V=800.0 PL=0
MOVL C00784 V=800.0 PL=0
MOVL C00785 V=800.0 PL=0
MOVL C00786 V=800.0 PL=0
MOVL C00787 V=800.0 PL=0
MOVL C00788 V=800.0 PL=0
MOVL C00789 V=800.0 PL=0
MOVL C00790 V=800.0 PL=0
MOVL C00791 V=800.0 PL=0
MOVL C00792 V=800.0 PL=0
MOVL C00793 V=800.0 PL=0
MOVL C00794 V=800.0 PL=0
MOVL C00795 V=800.0 PL=0
MOVL C00796 V=800.0 PL=0
MOVL C00797 V=800.0 PL=0
MOVL C00798 V=800.0 PL=0
MOVL C00799 V=800.0 PL=0
MOVL C00800 V=800.0 PL=0
MOVL C00801 V=800.0 PL=0
MOVL C00802 V=800.0 PL=0
MOVL C00803 V=800.0 PL=0
MOVL C00804 V=800.0 PL=0
MOVL C00805 V=800.0 PL=0
MOVL C00806 V=800.0 PL=0
MOVL C00807 V=800.0 PL=0
MOVL C00808 V=800.0 PL=0
MOVL C00809 V=800.0 PL=0
MOVL C00810 V=800.0 PL=0
MOVL C00811 V=800.0 PL=0
MOVL C00812 V=800.0 PL=0
MOVL C00813 V=800.0 PL=0
MOVL C00814 V=800.0 PL=0
MOVL C00815 V=800.0 PL=0
MOVL C00816 V=800.0 PL=0
MOVL C00817 V=800.0 PL=0
MOVL C00818 V=800.0 PL=0
MOVL C00819 V=800.0 PL=0
MOVL C00820 V=800.0 PL=0
MOVL C00821 V=800.0 PL=0
MOVL C00822 V=800.0 PL=0
MOVL C00823 V=800.0 PL=0
MOVL C00824 V=800.0 PL=0
MOVL C00825 V=800.0 PL=0
MOVL C00826 V=800.0 PL=0
MOVL C00827 V=800.0 PL=0
MOVL C00828 V=800.0 PL=0
MOVL C00829 V=800.0 PL=0
MOVL C00830 V=800.0 PL=0
MOVL C00831 V=800.0 PL=0
MOVL C00832 V=800.0 PL=0
MOVL C00833 V=800.0 PL=0
MOVL C00834 V=800.0 PL=0
MOVL C00835 V=800.0 PL=0
MOVL C00836 V=800.0 PL=0
MOVL C00837 V=800.0 PL=0
MOVL C00838 V=800.0 PL=0
MOVL C00839 V=800.0 PL=0
MOVL C00840 V=800.0 PL=0
MOVL C00841 V=800.0 PL=0
MOVL C00842 V=800.0 PL=0
MOVL C00843 V=800.0 PL=0
MOVL C00844 V=800.0 PL=0
MOVL C00845 V=800.0 PL=0
MOVL C00846 V=800.0 PL=0
MOVL C00847 V=800.0 PL=0
MOVL C00848 V=800.0 PL=0
MOVL C00849 V=800.0 PL=0
MOVL C00850 V=800.0 PL=0
MOVL C00851 V=800.0 PL=0
MOVL C00852 V=800.0 PL=0
MOVL C00853 V=800.0 PL=0
MOVL C00854 V=800.0 PL=0
MOVL C00855 V=800.0 PL=0
MOVL C00856 V=800.0 PL=0
MOVL C00857 V=800.0 PL=0
MOVL C00858 V=800.0 PL=0
MOVL C00859 V=800.0 PL=0
MOVL C00860 V=800.0 PL=0
MOVL C00861 V=800.0 PL=0
MOVL C00862 V=800.0 PL=0
MOVL C00863 V=800.0 PL=0
MOVL C00864 V=800.0 PL=0
MOVL C00865 V=800.0 PL=0
MOVL C00866 V=800.0 PL=0
MOVL C00867 V=800.0 PL=0
MOVL C00868 V=800.0 PL=0
MOVL C00869 V=800.0 PL=0
MOVL C00870 V=800.0 PL=0
MOVL C00871 V=800.0 PL=0
MOVL C00872 V=800.0 PL=0
MOVL C00873 V=800.0 PL=0
MOVL C00874 V=800.0 PL=0
MOVL C00875 V=800.0 PL=0
MOVL C00876 V=800.0 PL=0
MOVL C00877 V=800.0 PL=0
MOVL C00878 V=800.0 PL=0
MOVL C00879 V=800.0 PL=0
MOVL C00880 V=800.0 PL=0
MOVL C00881 V=800.0 PL=0
MOVL C00882 V=800.0 PL=0
MOVL C00883 V=800.0 PL=0
MOVL C00884 V=800.0 PL=0
MOVL C00885 V=800.0 PL=0
MOVL C00886 V=800.0 PL=0
MOVL C00887 V=800.0 PL=0
MOVL C00888 V=800.0 PL=0
MOVL C00889 V=800.0 PL=0
MOVL C00890 V=800.0 PL=0
MOVL C00891 V=800.0 PL=0
MOVL C00892 V=800.0 PL=0
MOVL C00893 V=800.0 PL=0
MOVL C00894 V=800.0 PL=0
MOVL C00895 V=800.0 PL=0
MOVL C00896 V=800.0 PL=0
MOVL C00897 V=800.0 PL=0
MOVL C00898 V=800.0 PL=0
MOVL C00899 V=800.0 PL=0
MOVL C00900 V=800.0 PL=0
MOVL C00901 V=800.0 PL=0
MOVL C00902 V=800.0 PL=0
MOVL C00903 V=800.0 PL=0
MOVL C00904 V=800.0 PL=0
MOVL C00905 V=800.0 PL=0
MOVL C00906 V=800.0 PL=0
MOVL C00907 V=800.0 PL=0
MOVL C00908 V=800.0 PL=0
MOVL C00909 V=800.0 PL=0
MOVL C00910 V=800.0 PL=0
MOVL C00911 V=800.0 PL=0
MOVL C00912 V=800.0 PL=0
MOVL C00913 V=800.0 PL=0
MOVL C00914 V=800.0 PL=0
MOVL C00915 V=800.0 PL=0
MOVL C00916 V=800.0 PL=0
MOVL C00917 V=800.0 PL=0
MOVL C00918 V=800.0 PL=0
MOVL C00919 V=800.0 PL=0
MOVL C00920 V=800.0 PL=0
MOVL C00921 V=800.0 PL=0
MOVL C00922 V=800.0 PL=0
MOVL C00923 V=800.0 PL=0
MOVL C00924 V=800.0 PL=0
MOVL C00925 V=800.0 PL=0
MOVL C00926 V=800.0 PL=0
MOVL C00927 V=800.0 PL=0
MOVL C00928 V=800.0 PL=0
MOVL C00929 V=800.0 PL=0
MOVL C00930 V=800.0 PL=0
MOVL C00931 V=800.0 PL=0
MOVL C00932 V=800.0 PL=0
MOVL C00933 V=800.0 PL=0
MOVL C00934 V=800.0 PL=0
MOVL C00935 V=800.0 PL=0
MOVL C00936 V=800.0 PL=0
MOVL C00937 V=800.0 PL=0
MOVL C00938 V=800.0 PL=0
MOVL C00939 V=800.0 PL=0
MOVL C00940 V=800.0 PL=0
MOVL C00941 V=800.0 PL=0
MOVL C00942 V=800.0 PL=0
MOVL C00943 V=800.0 PL=0
MOVL C00944 V=800.0 PL=0
MOVL C00945 V=800.0 PL=0
MOVL C00946 V=800.0 PL=0
MOVL C00947 V=800.0 PL=0
MOVL C00948 V=800.0 PL=0
MOVL C00949 V=800.0 PL=0
MOVL C00950 V=800.0 PL=0
MOVL C00951 V=800.0 PL=0
MOVL C00952 V=800.0 PL=0
MOVL C00953 V=800.0 PL=0
MOVL C00954 V=800.0 PL=0
MOVL C00955 V=800.0 PL=0
MOVL C00956 V=800.0 PL=0
MOVL C00957 V=800.0 PL=0
MOVL C00958 V=800.0 PL=0
MOVL C00959 V=800.0 PL=0
MOVL C00960 V=800.0 PL=0
MOVL C00961 V=800.0 PL=0
MOVL C00962 V=800.0 PL=0
MOVL C00963 V=800.0 PL=0
MOVL C00964 V=800.0 PL=0
MOVL C00965 V=800.0 PL=0
MOVL C00966 V=800.0 PL=0
MOVL C00967 V=800.0 PL=0
MOVL C00968 V=800.0 PL=0
MOVL C00969 V=800.0 PL=0
MOVL C00970 V=800.0 PL=0
MOVL C00971 V=800.0 PL=0
MOVL C00972 V=800.0 PL=0
MOVL C00973 V=800.0 PL=0
MOVL C00974 V=800.0 PL=0
MOVL C00975 V=800.0 PL=0
MOVL C00976 V=800.0 PL=0
MOVL C00977 V=800.0 PL=0
MOVL C00978 V=800.0 PL=0
MOVL C00979 V=800.0 PL=0
MOVL C00980 V=800.0 PL=0
MOVL C00981 V=800.0 PL=0
MOVL C00982 V=800.0 PL=0
MOVL C00983 V=800.0 PL=0
MOVL C00984 V=800.0 PL=0
MOVL C00985 V=800.0 PL=0
MOVL C00986 V=800.0 PL=0
MOVL C00987 V=800.0 PL=0
MOVL C00988 V=800.0 PL=0
MOVL C00989 V=800.0 PL=0
MOVL C00990 V=800.0 PL=0
MOVL C00991 V=800.0 PL=0
MOVL C00992 V=800.0 PL=0
MOVL C00993 V=800.0 PL=0
MOVL C00994 V=800.0 PL=0
MOVL C00995 V=800.0 PL=0
MOVL C00996 V=800.0 PL=0
MOVL C00997 V=800.0 PL=0
MOVL C00998 V=800.0 PL=0
MOVL C00999 V=800.0 PL=0
MOVL C01000 V=800.0 PL=0
MOVL C01001 V=800.0 PL=0
MOVL C01002 V=800.0 PL=0
MOVL C01003 V=800.0 PL=0
MOVL C01004 V=800.0 PL=0
MOVL C01005 V=800.0 PL=0
MOVL C01006 V=800.0 PL=0
MOVL C01007 V=800.0 PL=0
MOVL C01008 V=800.0 PL=0
MOVL C01009 V=800.0 PL=0
MOVL C01010 V=800.0 PL=0
MOVL C01011 V=800.0 PL=0
MOVL C01012 V=800.0 PL=0
MOVL C01013 V=800.0 PL=0
MOVL C01014 V=800.0 PL=0
MOVL C01015 V=800.0 PL=0
MOVL C01016 V=800.0 PL=0
MOVL C01017 V=800.0 PL=0
MOVL C01018 V=800.0 PL=0
MOVL C01019 V=800.0 PL=0
MOVL C01020 V=800.0 PL=0
MOVL C01021 V=800.0 PL=0
MOVL C01022 V=800.0 PL=0
MOVL C01023 V=800.0 PL=0
MOVL C01024 V=800.0 PL=0
MOVL C01025 V=800.0 PL=0
MOVL C01026 V=800.0 PL=0
MOVL C01027 V=800.0 PL=0
MOVL C01028 V=800.0 PL=0
MOVL C01029 V=800.0 PL=0
MOVL C01030 V=800.0 PL=0
MOVL C01031 V=800.0 PL=0
MOVL C01032 V=800.0 PL=0
MOVL C01033 V=800.0 PL=0
MOVL C01034 V=800.0 PL=0
MOVL C01035 V=800.0 PL=0
MOVL C01036 V=800.0 PL=0
MOVL C01037 V=800.0 PL=0
MOVL C01038 V=800.0 PL=0
MOVL C01039 V=800.0 PL=0
MOVL C01040 V=800.0 PL=0
MOVL C01041 V=800.0 PL=0
MOVL C01042 V=800.0 PL=0
MOVL C01043 V=800.0 PL=0
MOVL C01044 V=800.0 PL=0
MOVL C01045 V=800.0 PL=0
MOVL C01046 V=800.0 PL=0
MOVL C01047 V=800.0 PL=0
MOVL C01048 V=800.0 PL=0
MOVL C01049 V=800.0 PL=0
MOVL C01050 V=800.0 PL=0
MOVL C01051 V=800.0 PL=0
MOVL C01052 V=800.0 PL=0
MOVL C01053 V=800.0 PL=0
MOVL C01054 V=800.0 PL=0
MOVL C01055 V=800.0 PL=0
MOVL C01056 V=800.0 PL=0
MOVL C01057 V=800.0 PL=0
MOVL C01058 V=800.0 PL=0
MOVL C01059 V=800.0 PL=0
MOVL C01060 V=800.0 PL=0
MOVL C01061 V=800.0 PL=0
MOVL C01062 V=800.0 PL=0
MOVL C01063 V=800.0 PL=0
MOVL C01064 V=800.0 PL=0
MOVL C01065 V=800.0 PL=0
MOVL C01066 V=800.0 PL=0
MOVL C01067 V=800.0 PL=0
MOVL C01068 V=800.0 PL=0
MOVL C01069 V=800.0 PL=0
MOVL C01070 V=800.0 PL=0
MOVL C01071 V=800.0 PL=0
MOVL C01072 V=800.0 PL=0
MOVL C01073 V=800.0 PL=0
MOVL C01074 V=800.0 PL=0
MOVL C01075 V=800.0 PL=0
MOVL C01076 V=800.0 PL=0
MOVL C01077 V=800.0 PL=0
MOVL C01078 V=800.0 PL=0
MOVL C01079 V=800.0 PL=0
MOVL C01080 V=800.0 PL=0
MOVL C01081 V=800.0 PL=0
MOVL C01082 V=800.0 PL=0
MOVL C01083 V=800.0 PL=0
MOVL C01084 V=800.0 PL=0
MOVL C01085 V=800.0 PL=0
MOVL C01086 V=800.0 PL=0
MOVL C01087 V=800.0 PL=0
MOVL C01088 V=800.0 PL=0
MOVL C01089 V=800.0 PL=0
MOVL C01090 V=800.0 PL=0
MOVL C01091 V=800.0 PL=0
MOVL C01092 V=800.0 PL=0
MOVL C01093 V=800.0 PL=0
MOVL C01094 V=800.0 PL=0
MOVL C01095 V=800.0 PL=0
MOVL C01096 V=800.0 PL=0
MOVL C01097 V=800.0 PL=0
MOVL C01098 V=800.0 PL=0
MOVL C01099 V=800.0 PL=0
MOVL C01100 V=800.0 PL=0
MOVL C01101 V=800.0 PL=0
MOVL C01102 V=800.0 PL=0
MOVL C01103 V=800.0 PL=0
MOVL C01104 V=800.0 PL=0
MOVL C01105 V=800.0 PL=0
MOVL C01106 V=800.0 PL=0
MOVL C01107 V=800.0 PL=0
MOVL C01108 V=800.0 PL=0
MOVL C01109 V=800.0 PL=0
MOVL C01110 V=800.0 PL=0
MOVL C01111 V=800.0 PL=0
MOVL C01112 V=800.0 PL=0
MOVL C01113 V=800.0 PL=0
MOVL C01114 V=800.0 PL=0
MOVL C01115 V=800.0 PL=0
MOVL C01116 V=800.0 PL=0
MOVL C01117 V=800.0 PL=0
MOVL C01118 V=800.0 PL=0
MOVL C01119 V=800.0 PL=0
MOVL C01120 V=800.0 PL=0
MOVL C01121 V=800.0 PL=0
MOVL C01122 V=800.0 PL=0
MOVL C01123 V=800.0 PL=0
MOVL C01124 V=800.0 PL=0
MOVL C01125 V=800.0 PL=0
MOVL C01126 V=800.0 PL=0
MOVL C01127 V=800.0 PL=0
MOVL C01128 V=800.0 PL=0
MOVL C01129 V=800.0 PL=0
MOVL C01130 V=800.0 PL=0
MOVL C01131 V=800.0 PL=0
MOVL C01132 V=800.0 PL=0
MOVL C01133 V=800.0 PL=0
MOVL C01134 V=800.0 PL=0
MOVL C01135 V=800.0 PL=0
MOVL C01136 V=800.0 PL=0
MOVL C01137 V=800.0 PL=0
MOVL C01138 V=800.0 PL=0
MOVL C01139 V=800.0 PL=0
MOVL C01140 V=800.0 PL=0
MOVL C01141 V=800.0 PL=0
MOVL C01142 V=800.0 PL=0
MOVL C01143 V=800.0 PL=0
MOVL C01144 V=800.0 PL=0
MOVL C01145 V=800.0 PL=0
MOVL C01146 V=800.0 PL=0
MOVL C01147 V=800.0 PL=0
MOVL C01148 V=800.0 PL=0
MOVL C01149 V=800.0 PL=0
MOVL C01150 V=800.0 PL=0
MOVL C01151 V=800.0 PL=0
MOVL C01152 V=800.0 PL=0
MOVL C01153 V=800.0 PL=0
MOVL C01154 V=800.0 PL=0
MOVL C01155 V=800.0 PL=0
MOVL C01156 V=800.0 PL=0
MOVL C01157 V=800.0 PL=0
MOVL C01158 V=800.0 PL=0
MOVL C01159 V=800.0 PL=0
MOVL C01160 V=800.0 PL=0
MOVL C01161 V=800.0 PL=0
MOVL C01162 V=800.0 PL=0
MOVL C01163 V=800.0 PL=0
MOVL C01164 V=800.0 PL=0
MOVL C01165 V=800.0 PL=0
MOVL C01166 V=800.0 PL=0
MOVL C01167 V=800.0 PL=0
MOVL C01168 V=800.0 PL=0
MOVL C01169 V=800.0 PL=0
MOVL C01170 V=800.0 PL=0
MOVL C01171 V=800.0 PL=0
MOVL C01172 V=800.0 PL=0
MOVL C01173 V=800.0 PL=0
MOVL C01174 V=800.0 PL=0
MOVL C01175 V=800.0 PL=0
MOVL C01176 V=800.0 PL=0
MOVL C01177 V=800.0 PL=0
MOVL C01178 V=800.0 PL=0
MOVL C01179 V=800.0 PL=0
MOVL C01180 V=800.0 PL=0
MOVL C01181 V=800.0 PL=0
MOVL C01182 V=800.0 PL=0
MOVL C01183 V=800.0 PL=0
MOVL C01184 V=800.0 PL=0
MOVL C01185 V=800.0 PL=0
MOVL C01186 V=800.0 PL=0
MOVL C01187 V=800.0 PL=0
MOVL C01188 V=800.0 PL=0
MOVL C01189 V=800.0 PL=0
MOVL C01190 V=800.0 PL=0
MOVL C01191 V=800.0 PL=0
MOVL C01192 V=800.0 PL=0
MOVL C01193 V=800.0 PL=0
MOVL C01194 V=800.0 PL=0
MOVL C01195 V=800.0 PL=0
MOVL C01196 V=800.0 PL=0
MOVL C01197 V=800.0 PL=0
MOVL C01198 V=800.0 PL=0
MOVL C01199 V=800.0 PL=0
MOVL C01200 V=800.0 PL=0
MOVL C01201 V=800.0 PL=0
MOVL C01202 V=800.0 PL=0
MOVL C01203 V=800.0 PL=0
MOVL C01204 V=800.0 PL=0
MOVL C01205 V=800.0 PL=0
MOVL C01206 V=800.0 PL=0
MOVL C01207 V=800.0 PL=0
MOVL C01208 V=800.0 PL=0
MOVL C01209 V=800.0 PL=0
MOVL C01210 V=800.0 PL=0
MOVL C01211 V=800.0 PL=0
MOVL C01212 V=800.0 PL=0
MOVL C01213 V=800.0 PL=0
MOVL C01214 V=800.0 PL=0
MOVL C01215 V=800.0 PL=0
MOVL C01216 V=800.0 PL=0
MOVL C01217 V=800.0 PL=0
MOVL C01218 V=800.0 PL=0
MOVL C01219 V=800.0 PL=0
MOVL C01220 V=800.0 PL=0
MOVL C01221 V=800.0 PL=0
MOVL C01222 V=800.0 PL=0
MOVL C01223 V=800.0 PL=0
MOVL C01224 V=800.0 PL=0
MOVL C01225 V=800.0 PL=0
MOVL C01226 V=800.0 PL=0
MOVL C01227 V=800.0 PL=0
MOVL C01228 V=800.0 PL=0
MOVL C01229 V=800.0 PL=0
MOVL C01230 V=800.0 PL=0
MOVL C01231 V=800.0 PL=0
MOVL C01232 V=800.0 PL=0
MOVL C01233 V=800.0 PL=0
MOVL C01234 V=800.0 PL=0
MOVL C01235 V=800.0 PL=0
MOVL C01236 V=800.0 PL=0
MOVL C01237 V=800.0 PL=0
MOVL C01238 V=800.0 PL=0
MOVL C01239 V=800.0 PL=0
MOVL C01240 V=800.0 PL=0
MOVL C01241 V=800.0 PL=0
MOVL C01242 V=800.0 PL=0
MOVL C01243 V=800.0 PL=0
MOVL C01244 V=800.0 PL=0
MOVL C01245 V=800.0 PL=0
MOVL C01246 V=800.0 PL=0
MOVL C01247 V=800.0 PL=0
MOVL C01248 V=800.0 PL=0
MOVL C01249 V=800.0 PL=0
MOVL C01250 V=800.0 PL=0
MOVL C01251 V=800.0 PL=0
MOVL C01252 V=800.0 PL=0
MOVL C01253 V=800.0 PL=0
MOVL C01254 V=800.0 PL=0
MOVL C01255 V=800.0 PL=0
MOVL C01256 V=800.0 PL=0
MOVL C01257 V=800.0 PL=0
MOVL C01258 V=800.0 PL=0
MOVL C01259 V=800.0 PL=0
MOVL C01260 V=800.0 PL=0
MOVL C01261 V=800.0 PL=0
MOVL C01262 V=800.0 PL=0
MOVL C01263 V=800.0 PL=0
MOVL C01264 V=800.0 PL=0
MOVL C01265 V=800.0 PL=0
MOVL C01266 V=800.0 PL=0
MOVL C01267 V=800.0 PL=0
MOVL C01268 V=800.0 PL=0
MOVL C01269 V=800.0 PL=0
MOVL C01270 V=800.0 PL=0
MOVL C01271 V=800.0 PL=0
MOVL C01272 V=800.0 PL=0
MOVL C01273 V=800.0 PL=0
MOVL C01274 V=800.0 PL=0
MOVL C01275 V=800.0 PL=0
MOVL C01276 V=800.0 PL=0
MOVL C01277 V=800.0 PL=0
MOVL C01278 V=800.0 PL=0
MOVL C01279 V=800.0 PL=0
MOVL C01280 V=800.0 PL=0
MOVL C01281 V=800.0 PL=0
MOVL C01282 V=800.0 PL=0
MOVL C01283 V=800.0 PL=0
MOVL C01284 V=800.0 PL=0
MOVL C01285 V=800.0 PL=0
MOVL C01286 V=800.0 PL=0
MOVL C01287 V=800.0 PL=0
MOVL C01288 V=800.0 PL=0
MOVL C01289 V=800.0 PL=0
MOVL C01290 V=800.0 PL=0
MOVL C01291 V=800.0 PL=0
MOVL C01292 V=800.0 PL=0
MOVL C01293 V=800.0 PL=0
MOVL C01294 V=800.0 PL=0
MOVL C01295 V=800.0 PL=0
MOVL C01296 V=800.0 PL=0
MOVL C01297 V=800.0 PL=0
MOVL C01298 V=800.0 PL=0
MOVL C01299 V=800.0 PL=0
MOVL C01300 V=800.0 PL=0
MOVL C01301 V=800.0 PL=0
MOVL C01302 V=800.0 PL=0
MOVL C01303 V=800.0 PL=0
MOVL C01304 V=800.0 PL=0
MOVL C01305 V=800.0 PL=0
MOVL C01306 V=800.0 PL=0
MOVL C01307 V=800.0 PL=0
MOVL C01308 V=800.0 PL=0
MOVL C01309 V=800.0 PL=0
MOVL C01310 V=800.0 PL=0
MOVL C01311 V=800.0 PL=0
MOVL C01312 V=800.0 PL=0
MOVL C01313 V=800.0 PL=0
MOVL C01314 V=800.0 PL=0
MOVL C01315 V=800.0 PL=0
MOVL C01316 V=800.0 PL=0
MOVL C01317 V=800.0 PL=0
MOVL C01318 V=800.0 PL=0
MOVL C01319 V=800.0 PL=0
MOVL C01320 V=800.0 PL=0
MOVL C01321 V=800.0 PL=0
MOVL C01322 V=800.0 PL=0
MOVL C01323 V=800.0 PL=0
MOVL C01324 V=800.0 PL=0
MOVL C01325 V=800.0 PL=0
MOVL C01326 V=800.0 PL=0
MOVL C01327 V=800.0 PL=0
MOVL C01328 V=800.0 PL=0
MOVL C01329 V=800.0 PL=0
MOVL C01330 V=800.0 PL=0
MOVL C01331 V=800.0 PL=0
MOVL C01332 V=800.0 PL=0
MOVL C01333 V=800.0 PL=0
MOVL C01334 V=800.0 PL=0
MOVL C01335 V=800.0 PL=0
MOVL C01336 V=800.0 PL=0
MOVL C01337 V=800.0 PL=0
MOVL C01338 V=800.0 PL=0
MOVL C01339 V=800.0 PL=0
MOVL C01340 V=800.0 PL=0
MOVL C01341 V=800.0 PL=0
MOVL C01342 V=800.0 PL=0
MOVL C01343 V=800.0 PL=0
MOVL C01344 V=800.0 PL=0
MOVL C01345 V=800.0 PL=0
MOVL C01346 V=800.0 PL=0
MOVL C01347 V=800.0 PL=0
MOVL C01348 V=800.0 PL=0
MOVL C01349 V=800.0 PL=0
MOVL C01350 V=800.0 PL=0
MOVL C01351 V=800.0 PL=0
MOVL C01352 V=800.0 PL=0
MOVL C01353 V=800.0 PL=0
MOVL C01354 V=800.0 PL=0
MOVL C01355 V=800.0 PL=0
MOVL C01356 V=800.0 PL=0
MOVL C01357 V=800.0 PL=0
MOVL C01358 V=800.0 PL=0
MOVL C01359 V=800.0 PL=0
MOVL C01360 V=800.0 PL=0
MOVL C01361 V=800.0 PL=0
MOVL C01362 V=800.0 PL=0
MOVL C01363 V=800.0 PL=0
MOVL C01364 V=800.0 PL=0
MOVL C01365 V=800.0 PL=0
MOVL C01366 V=800.0 PL=0
MOVL C01367 V=800.0 PL=0
MOVL C01368 V=800.0 PL=0
MOVL C01369 V=800.0 PL=0
MOVL C01370 V=800.0 PL=0
MOVL C01371 V=800.0 PL=0
MOVL C01372 V=800.0 PL=0
MOVL C01373 V=800.0 PL=0
MOVL C01374 V=800.0 PL=0
MOVL C01375 V=800.0 PL=0
MOVL C01376 V=800.0 PL=0
MOVL C01377 V=800.0 PL=0
MOVL C01378 V=800.0 PL=0
MOVL C01379 V=800.0 PL=0
MOVL C01380 V=800.0 PL=0
MOVL C01381 V=800.0 PL=0
MOVL C01382 V=800.0 PL=0
MOVL C01383 V=800.0 PL=0
MOVL C01384 V=800.0 PL=0
MOVL C01385 V=800.0 PL=0
MOVL C01386 V=800.0 PL=0
MOVL C01387 V=800.0 PL=0
MOVL C01388 V=800.0 PL=0
MOVL C01389 V=800.0 PL=0
MOVL C01390 V=800.0 PL=0
MOVL C01391 V=800.0 PL=0
MOVL C01392 V=800.0 PL=0
MOVL C01393 V=800.0 PL=0
MOVL C01394 V=800.0 PL=0
MOVL C01395 V=800.0 PL=0
MOVL C01396 V=800.0 PL=0
MOVL C01397 V=800.0 PL=0
MOVL C01398 V=800.0 PL=0
MOVL C01399 V=800.0 PL=0
MOVL C01400 V=800.0 PL=0
MOVL C01401 V=800.0 PL=0
MOVL C01402 V=800.0 PL=0
MOVL C01403 V=800.0 PL=0
MOVL C01404 V=800.0 PL=0
MOVL C01405 V=800.0 PL=0
MOVL C01406 V=800.0 PL=0
MOVL C01407 V=800.0 PL=0
MOVL C01408 V=800.0 PL=0
MOVL C01409 V=800.0 PL=0
MOVL C01410 V=800.0 PL=0
MOVL C01411 V=800.0 PL=0
MOVL C01412 V=800.0 PL=0
MOVL C01413 V=800.0 PL=0
MOVL C01414 V=800.0 PL=0
MOVL C01415 V=800.0 PL=0
MOVL C01416 V=800.0 PL=0
MOVL C01417 V=800.0 PL=0
MOVL C01418 V=800.0 PL=0
MOVL C01419 V=800.0 PL=0
MOVL C01420 V=800.0 PL=0
MOVL C01421 V=800.0 PL=0
MOVL C01422 V=800.0 PL=0
MOVL C01423 V=800.0 PL=0
MOVL C01424 V=800.0 PL=0
MOVL C01425 V=800.0 PL=0
MOVL C01426 V=800.0 PL=0
MOVL C01427 V=800.0 PL=0
MOVL C01428 V=800.0 PL=0
MOVL C01429 V=800.0 PL=0
MOVL C01430 V=800.0 PL=0
MOVL C01431 V=800.0 PL=0
MOVL C01432 V=800.0 PL=0
MOVL C01433 V=800.0 PL=0
MOVL C01434 V=800.0 PL=0
MOVL C01435 V=800.0 PL=0
MOVL C01436 V=800.0 PL=0
MOVL C01437 V=800.0 PL=0
MOVL C01438 V=800.0 PL=0
MOVL C01439 V=800.0 PL=0
MOVL C01440 V=800.0 PL=0
MOVL C01441 V=800.0 PL=0
MOVL C01442 V=800.0 PL=0
MOVL C01443 V=800.0 PL=0
MOVL C01444 V=800.0 PL=0
MOVL C01445 V=800.0 PL=0
MOVL C01446 V=800.0 PL=0
MOVL C01447 V=800.0 PL=0
MOVL C01448 V=800.0 PL=0
MOVL C01449 V=800.0 PL=0
MOVL C01450 V=800.0 PL=0
MOVL C01451 V=800.0 PL=0
MOVL C01452 V=800.0 PL=0
MOVL C01453 V=800.0 PL=0
MOVL C01454 V=800.0 PL=0
MOVL C01455 V=800.0 PL=0
MOVL C01456 V=800.0 PL=0
MOVL C01457 V=800.0 PL=0
MOVL C01458 V=800.0 PL=0
MOVL C01459 V=800.0 PL=0
MOVL C01460 V=800.0 PL=0
MOVL C01461 V=800.0 PL=0
MOVL C01462 V=800.0 PL=0
MOVL C01463 V=800.0 PL=0
MOVL C01464 V=800.0 PL=0
MOVL C01465 V=800.0 PL=0
MOVL C01466 V=800.0 PL=0
MOVL C01467 V=800.0 PL=0
MOVL C01468 V=800.0 PL=0
MOVL C01469 V=800.0 PL=0
MOVL C01470 V=800.0 PL=0
MOVL C01471 V=800.0 PL=0
MOVL C01472 V=800.0 PL=0
MOVL C01473 V=800.0 PL=0
MOVL C01474 V=800.0 PL=0
MOVL C01475 V=800.0 PL=0
MOVL C01476 V=800.0 PL=0
MOVL C01477 V=800.0 PL=0
MOVL C01478 V=800.0 PL=0
MOVL C01479 V=800.0 PL=0
MOVL C01480 V=800.0 PL=0
MOVL C01481 V=800.0 PL=0
MOVL C01482 V=800.0 PL=0
MOVL C01483 V=800.0 PL=0
MOVL C01484 V=800.0 PL=0
MOVL C01485 V=800.0 PL=0
MOVL C01486 V=800.0 PL=0
MOVL C01487 V=800.0 PL=0
MOVL C01488 V=800.0 PL=0
MOVL C01489 V=800.0 PL=0
MOVL C01490 V=800.0 PL=0
MOVL C01491 V=800.0 PL=0
MOVL C01492 V=800.0 PL=0
MOVL C01493 V=800.0 PL=0
MOVL C01494 V=800.0 PL=0
MOVL C01495 V=800.0 PL=0
MOVL C01496 V=800.0 PL=0
MOVL C01497 V=800.0 PL=0
MOVL C01498 V=800.0 PL=0
MOVL C01499 V=800.0 PL=0
MOVL C01500 V=800.0 PL=0
MOVL C01501 V=800.0 PL=0
MOVL C01502 V=800.0 PL=0
MOVL C01503 V=800.0 PL=0
MOVL C01504 V=800.0 PL=0
MOVL C01505 V=800.0 PL=0
MOVL C01506 V=800.0 PL=0
MOVL C01507 V=800.0 PL=0
MOVL C01508 V=800.0 PL=0
MOVL C01509 V=800.0 PL=0
MOVL C01510 V=800.0 PL=0
MOVL C01511 V=800.0 PL=0
MOVL C01512 V=800.0 PL=0
MOVL C01513 V=800.0 PL=0
MOVL C01514 V=800.0 PL=0
MOVL C01515 V=800.0 PL=0
MOVL C01516 V=800.0 PL=0
MOVL C01517 V=800.0 PL=0
MOVL C01518 V=800.0 PL=0
MOVL C01519 V=800.0 PL=0
MOVL C01520 V=800.0 PL=0
MOVL C01521 V=800.0 PL=0
MOVL C01522 V=800.0 PL=0
MOVL C01523 V=800.0 PL=0
MOVL C01524 V=800.0 PL=0
MOVL C01525 V=800.0 PL=0
MOVL C01526 V=800.0 PL=0
MOVL C01527 V=800.0 PL=0
MOVL C01528 V=800.0 PL=0
MOVL C01529 V=800.0 PL=0
MOVL C01530 V=800.0 PL=0
MOVL C01531 V=800.0 PL=0
MOVL C01532 V=800.0 PL=0
MOVL C01533 V=800.0 PL=0
MOVL C01534 V=800.0 PL=0
MOVL C01535 V=800.0 PL=0
MOVL C01536 V=800.0 PL=0
MOVL C01537 V=800.0 PL=0
MOVL C01538 V=800.0 PL=0
MOVL C01539 V=800.0 PL=0
MOVL C01540 V=800.0 PL=0
MOVL C01541 V=800.0 PL=0
MOVL C01542 V=800.0 PL=0
MOVL C01543 V=800.0 PL=0
MOVL C01544 V=800.0 PL=0
MOVL C01545 V=800.0 PL=0
MOVL C01546 V=800.0 PL=0
MOVL C01547 V=800.0 PL=0
MOVL C01548 V=800.0 PL=0
MOVL C01549 V=800.0 PL=0
MOVL C01550 V=800.0 PL=0
MOVL C01551 V=800.0 PL=0
MOVL C01552 V=800.0 PL=0
MOVL C01553 V=800.0 PL=0
MOVL C01554 V=800.0 PL=0
MOVL C01555 V=800.0 PL=0
MOVL C01556 V=800.0 PL=0
MOVL C01557 V=800.0 PL=0
MOVL C01558 V=800.0 PL=0
MOVL C01559 V=800.0 PL=0
MOVL C01560 V=800.0 PL=0
MOVL C01561 V=800.0 PL=0
MOVL C01562 V=800.0 PL=0
MOVL C01563 V=800.0 PL=0
MOVL C01564 V=800.0 PL=0
MOVL C01565 V=800.0 PL=0
MOVL C01566 V=800.0 PL=0
MOVL C01567 V=800.0 PL=0
MOVL C01568 V=800.0 PL=0
MOVL C01569 V=800.0 PL=0
MOVL C01570 V=800.0 PL=0
MOVL C01571 V=800.0 PL=0
MOVL C01572 V=800.0 PL=0
MOVL C01573 V=800.0 PL=0
MOVL C01574 V=800.0 PL=0
MOVL C01575 V=800.0 PL=0
MOVL C01576 V=800.0 PL=0
MOVL C01577 V=800.0 PL=0
MOVL C01578 V=800.0 PL=0
MOVL C01579 V=800.0 PL=0
MOVL C01580 V=800.0 PL=0
MOVL C01581 V=800.0 PL=0
MOVL C01582 V=800.0 PL=0
MOVL C01583 V=800.0 PL=0
MOVL C01584 V=800.0 PL=0
MOVL C01585 V=800.0 PL=0
MOVL C01586 V=800.0 PL=0
MOVL C01587 V=800.0 PL=0
MOVL C01588 V=800.0 PL=0
MOVL C01589 V=800.0 PL=0
MOVL C01590 V=800.0 PL=0
MOVL C01591 V=800.0 PL=0
MOVL C01592 V=800.0 PL=0
MOVL C01593 V=800.0 PL=0
MOVL C01594 V=800.0 PL=0
MOVL C01595 V=800.0 PL=0
MOVL C01596 V=800.0 PL=0
MOVL C01597 V=800.0 PL=0
MOVL C01598 V=800.0 PL=0
MOVL C01599 V=800.0 PL=0
MOVL C01600 V=800.0 PL=0
MOVL C01601 V=800.0 PL=0
MOVL C01602 V=800.0 PL=0
MOVL C01603 V=800.0 PL=0
MOVL C01604 V=800.0 PL=0
MOVL C01605 V=800.0 PL=0
MOVL C01606 V=800.0 PL=0
MOVL C01607 V=800.0 PL=0
MOVL C01608 V=800.0 PL=0
MOVL C01609 V=800.0 PL=0
MOVL C01610 V=800.0 PL=0
MOVL C01611 V=800.0 PL=0
MOVL C01612 V=800.0 PL=0
MOVL C01613 V=800.0 PL=0
MOVL C01614 V=800.0 PL=0
MOVL C01615 V=800.0 PL=0
MOVL C01616 V=800.0 PL=0
MOVL C01617 V=800.0 PL=0
MOVL C01618 V=800.0 PL=0
MOVL C01619 V=800.0 PL=0
MOVL C01620 V=800.0 PL=0
MOVL C01621 V=800.0 PL=0
MOVL C01622 V=800.0 PL=0
MOVL C01623 V=800.0 PL=0
MOVL C01624 V=800.0 PL=0
MOVL C01625 V=800.0 PL=0
MOVL C01626 V=800.0 PL=0
MOVL C01627 V=800.0 PL=0
MOVL C01628 V=800.0 PL=0
MOVL C01629 V=800.0 PL=0
MOVL C01630 V=800.0 PL=0
MOVL C01631 V=800.0 PL=0
MOVL C01632 V=800.0 PL=0
MOVL C01633 V=800.0 PL=0
MOVL C01634 V=800.0 PL=0
MOVL C01635 V=800.0 PL=0
MOVL C01636 V=800.0 PL=0
MOVL C01637 V=800.0 PL=0
MOVL C01638 V=800.0 PL=0
MOVL C01639 V=800.0 PL=0
MOVL C01640 V=800.0 PL=0
MOVL C01641 V=800.0 PL=0
MOVL C01642 V=800.0 PL=0
MOVL C01643 V=800.0 PL=0
MOVL C01644 V=800.0 PL=0
MOVL C01645 V=800.0 PL=0
MOVL C01646 V=800.0 PL=0
MOVL C01647 V=800.0 PL=0
MOVL C01648 V=800.0 PL=0
MOVL C01649 V=800.0 PL=0
MOVL C01650 V=800.0 PL=0
MOVL C01651 V=800.0 PL=0
MOVL C01652 V=800.0 PL=0
MOVL C01653 V=800.0 PL=0
MOVL C01654 V=800.0 PL=0
MOVL C01655 V=800.0 PL=0
MOVL C01656 V=800.0 PL=0
MOVL C01657 V=800.0 PL=0
MOVL C01658 V=800.0 PL=0
MOVL C01659 V=800.0 PL=0
MOVL C01660 V=800.0 PL=0
MOVL C01661 V=800.0 PL=0
MOVL C01662 V=800.0 PL=0
MOVL C01663 V=800.0 PL=0
MOVL C01664 V=800.0 PL=0
MOVL C01665 V=800.0 PL=0
MOVL C01666 V=800.0 PL=0
MOVL C01667 V=800.0 PL=0
MOVL C01668 V=800.0 PL=0
MOVL C01669 V=800.0 PL=0
MOVL C01670 V=800.0 PL=0
MOVL C01671 V=800.0 PL=0
MOVL C01672 V=800.0 PL=0
MOVL C01673 V=800.0 PL=0
MOVL C01674 V=800.0 PL=0
MOVL C01675 V=800.0 PL=0
MOVL C01676 V=800.0 PL=0
MOVL C01677 V=800.0 PL=0
MOVL C01678 V=800.0 PL=0
MOVL C01679 V=800.0 PL=0
MOVL C01680 V=800.0 PL=0
MOVL C01681 V=800.0 PL=0
MOVL C01682 V=800.0 PL=0
MOVL C01683 V=800.0 PL=0
MOVL C01684 V=800.0 PL=0
MOVL C01685 V=800.0 PL=0
MOVL C01686 V=800.0 PL=0
MOVL C01687 V=800.0 PL=0
MOVL C01688 V=800.0 PL=0
MOVL C01689 V=800.0 PL=0
MOVL C01690 V=800.0 PL=0
MOVL C01691 V=800.0 PL=0
MOVL C01692 V=800.0 PL=0
MOVL C01693 V=800.0 PL=0
MOVL C01694 V=800.0 PL=0
MOVL C01695 V=800.0 PL=0
MOVL C01696 V=800.0 PL=0
MOVL C01697 V=800.0 PL=0
MOVL C01698 V=800.0 PL=0
MOVL C01699 V=800.0 PL=0
MOVL C01700 V=800.0 PL=0
MOVL C01701 V=800.0 PL=0
MOVL C01702 V=800.0 PL=0
MOVL C01703 V=800.0 PL=0
MOVL C01704 V=800.0 PL=0
MOVL C01705 V=800.0 PL=0
MOVL C01706 V=800.0 PL=0
MOVL C01707 V=800.0 PL=0
MOVL C01708 V=800.0 PL=0
MOVL C01709 V=800.0 PL=0
MOVL C01710 V=800.0 PL=0
MOVL C01711 V=800.0 PL=0
MOVL C01712 V=800.0 PL=0
MOVL C01713 V=800.0 PL=0
MOVL C01714 V=800.0 PL=0
MOVL C01715 V=800.0 PL=0
MOVL C01716 V=800.0 PL=0
MOVL C01717 V=800.0 PL=0
MOVL C01718 V=800.0 PL=0
MOVL C01719 V=800.0 PL=0
MOVL C01720 V=800.0 PL=0
MOVL C01721 V=800.0 PL=0
MOVL C01722 V=800.0 PL=0
MOVL C01723 V=800.0 PL=0
MOVL C01724 V=800.0 PL=0
MOVL C01725 V=800.0 PL=0
MOVL C01726 V=800.0 PL=0
MOVL C01727 V=800.0 PL=0
MOVL C01728 V=800.0 PL=0
MOVL C01729 V=800.0 PL=0
MOVL C01730 V=800.0 PL=0
MOVL C01731 V=800.0 PL=0
MOVL C01732 V=800.0 PL=0
MOVL C01733 V=800.0 PL=0
MOVL C01734 V=800.0 PL=0
MOVL C01735 V=800.0 PL=0
MOVL C01736 V=800.0 PL=0
MOVL C01737 V=800.0 PL=0
MOVL C01738 V=800.0 PL=0
MOVL C01739 V=800.0 PL=0
MOVL C01740 V=800.0 PL=0
MOVL C01741 V=800.0 PL=0
MOVL C01742 V=800.0 PL=0
MOVL C01743 V=800.0 PL=0
MOVL C01744 V=800.0 PL=0
MOVL C01745 V=800.0 PL=0
MOVL C01746 V=800.0 PL=0
MOVL C01747 V=800.0 PL=0
MOVL C01748 V=800.0 PL=0
MOVL C01749 V=800.0 PL=0
MOVL C01750 V=800.0 PL=0
MOVL C01751 V=800.0 PL=0
MOVL C01752 V=800.0 PL=0
MOVL C01753 V=800.0 PL=0
MOVL C01754 V=800.0 PL=0
MOVL C01755 V=800.0 PL=0
MOVL C01756 V=800.0 PL=0
MOVL C01757 V=800.0 PL=0
MOVL C01758 V=800.0 PL=0
MOVL C01759 V=800.0 PL=0
MOVL C01760 V=800.0 PL=0
MOVL C01761 V=800.0 PL=0
MOVL C01762 V=800.0 PL=0
MOVL C01763 V=800.0 PL=0
MOVL C01764 V=800.0 PL=0
MOVL C01765 V=800.0 PL=0
MOVL C01766 V=800.0 PL=0
MOVL C01767 V=800.0 PL=0
MOVL C01768 V=800.0 PL=0
MOVL C01769 V=800.0 PL=0
MOVL C01770 V=800.0 PL=0
MOVL C01771 V=800.0 PL=0
MOVL C01772 V=800.0 PL=0
MOVL C01773 V=800.0 PL=0
MOVL C01774 V=800.0 PL=0
MOVL C01775 V=800.0 PL=0
MOVL C01776 V=800.0 PL=0
MOVL C01777 V=800.0 PL=0
MOVL C01778 V=800.0 PL=0
MOVL C01779 V=800.0 PL=0
MOVL C01780 V=800.0 PL=0
MOVL C01781 V=800.0 PL=0
MOVL C01782 V=800.0 PL=0
MOVL C01783 V=800.0 PL=0
MOVL C01784 V=800.0 PL=0
MOVL C01785 V=800.0 PL=0
MOVL C01786 V=800.0 PL=0
MOVL C01787 V=800.0 PL=0
MOVL C01788 V=800.0 PL=0
MOVL C01789 V=800.0 PL=0
MOVL C01790 V=800.0 PL=0
MOVL C01791 V=800.0 PL=0
MOVL C01792 V=800.0 PL=0
MOVL C01793 V=800.0 PL=0
MOVL C01794 V=800.0 PL=0
MOVL C01795 V=800.0 PL=0
MOVL C01796 V=800.0 PL=0
MOVL C01797 V=800.0 PL=0
MOVL C01798 V=800.0 PL=0
MOVL C01799 V=800.0 PL=0
MOVL C01800 V=800.0 PL=0
MOVL C01801 V=800.0 PL=0
MOVL C01802 V=800.0 PL=0
MOVL C01803 V=800.0 PL=0
MOVL C01804 V=800.0 PL=0
MOVL C01805 V=800.0 PL=0
MOVL C01806 V=800.0 PL=0
MOVL C01807 V=800.0 PL=0
MOVL C01808 V=800.0 PL=0
MOVL C01809 V=800.0 PL=0
MOVL C01810 V=800.0 PL=0
MOVL C01811 V=800.0 PL=0
MOVL C01812 V=800.0 PL=0
MOVL C01813 V=800.0 PL=0
MOVL C01814 V=800.0 PL=0
MOVL C01815 V=800.0 PL=0
MOVL C01816 V=800.0 PL=0
MOVL C01817 V=800.0 PL=0
MOVL C01818 V=800.0 PL=0
MOVL C01819 V=800.0 PL=0
MOVL C01820 V=800.0 PL=0
MOVL C01821 V=800.0 PL=0
MOVL C01822 V=800.0 PL=0
MOVL C01823 V=800.0 PL=0
MOVL C01824 V=800.0 PL=0
MOVL C01825 V=800.0 PL=0
MOVL C01826 V=800.0 PL=0
MOVL C01827 V=800.0 PL=0
MOVL C01828 V=800.0 PL=0
MOVL C01829 V=800.0 PL=0
MOVL C01830 V=800.0 PL=0
MOVL C01831 V=800.0 PL=0
MOVL C01832 V=800.0 PL=0
MOVL C01833 V=800.0 PL=0
MOVL C01834 V=800.0 PL=0
MOVL C01835 V=800.0 PL=0
MOVL C01836 V=800.0 PL=0
MOVL C01837 V=800.0 PL=0
MOVL C01838 V=800.0 PL=0
MOVL C01839 V=800.0 PL=0
MOVL C01840 V=800.0 PL=0
MOVL C01841 V=800.0 PL=0
MOVL C01842 V=800.0 PL=0
MOVL C01843 V=800.0 PL=0
MOVL C01844 V=800.0 PL=0
MOVL C01845 V=800.0 PL=0
MOVL C01846 V=800.0 PL=0
MOVL C01847 V=800.0 PL=0
MOVL C01848 V=800.0 PL=0
MOVL C01849 V=800.0 PL=0
MOVL C01850 V=800.0 PL=0
MOVL C01851 V=800.0 PL=0
MOVL C01852 V=800.0 PL=0
MOVL C01853 V=800.0 PL=0
MOVL C01854 V=800.0 PL=0
MOVL C01855 V=800.0 PL=0
MOVL C01856 V=800.0 PL=0
MOVL C01857 V=800.0 PL=0
MOVL C01858 V=800.0 PL=0
MOVL C01859 V=800.0 PL=0
MOVL C01860 V=800.0 PL=0
MOVL C01861 V=800.0 PL=0
MOVL C01862 V=800.0 PL=0
MOVL C01863 V=800.0 PL=0
MOVL C01864 V=800.0 PL=0
MOVL C01865 V=800.0 PL=0
MOVL C01866 V=800.0 PL=0
MOVL C01867 V=800.0 PL=0
MOVL C01868 V=800.0 PL=0
MOVL C01869 V=800.0 PL=0
MOVL C01870 V=800.0 PL=0
MOVL C01871 V=800.0 PL=0
MOVL C01872 V=800.0 PL=0
MOVL C01873 V=800.0 PL=0
MOVL C01874 V=800.0 PL=0
MOVL C01875 V=800.0 PL=0
MOVL C01876 V=800.0 PL=0
MOVL C01877 V=800.0 PL=0
MOVL C01878 V=800.0 PL=0
MOVL C01879 V=800.0 PL=0
MOVL C01880 V=800.0 PL=0
MOVL C01881 V=800.0 PL=0
MOVL C01882 V=800.0 PL=0
MOVL C01883 V=800.0 PL=0
MOVL C01884 V=800.0 PL=0
MOVL C01885 V=800.0 PL=0
MOVL C01886 V=800.0 PL=0
MOVL C01887 V=800.0 PL=0
MOVL C01888 V=800.0 PL=0
MOVL C01889 V=800.0 PL=0
MOVL C01890 V=800.0 PL=0
MOVL C01891 V=800.0 PL=0
MOVL C01892 V=800.0 PL=0
MOVL C01893 V=800.0 PL=0
MOVL C01894 V=800.0 PL=0
MOVL C01895 V=800.0 PL=0
MOVL C01896 V=800.0 PL=0
MOVL C01897 V=800.0 PL=0
MOVL C01898 V=800.0 PL=0
MOVL C01899 V=800.0 PL=0
MOVL C01900 V=800.0 PL=0
MOVL C01901 V=800.0 PL=0
MOVL C01902 V=800.0 PL=0
MOVL C01903 V=800.0 PL=0
MOVL C01904 V=800.0 PL=0
MOVL C01905 V=800.0 PL=0
MOVL C01906 V=800.0 PL=0
